KUKA KRL program: EPS_2_25862_MH4A_A_20251016034300.src

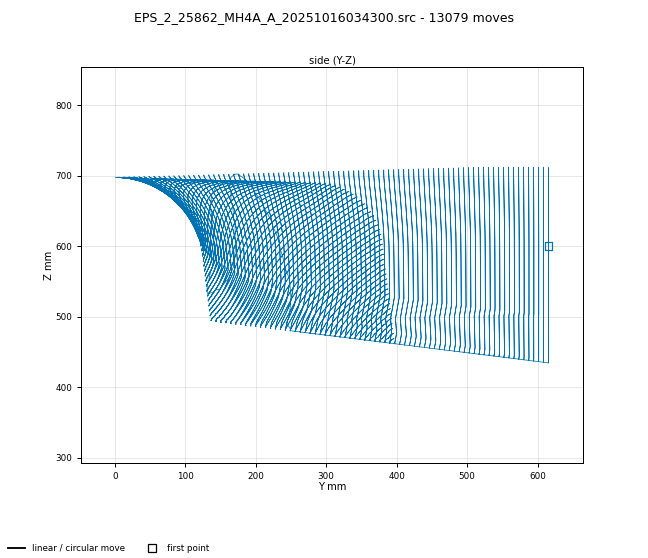
[picture p0: tool path of EPS_2_25862_MH4A_A_20251016034300.src, 13079 of 13081 moves have a stored position in this frame; points joined in program order, loops and branches not executed]
&ACCESS RVP
&REL 4
&COMMENT QRS 19112012
&PARAM EDITMASK = *
DEF PART()
EXT BAS (BAS_COMMAND :IN,REAL :IN )
INT I
BAS (#INITMOV,0 )

;KUKA QRS Post kuka4.cps  Date:22-06-2017 !

File_ID=2890

QRS_PRE_INIT()

;Init var - Until changes are made in qrs_pre_init
Outlet_Square_prg=0
Inlet_1_Square_prg=0
Inlet_2_Square_prg=0
Inlet_3_Square_prg=0
Inlet_4_Square_prg=0
Inlet_5_Square_prg=0

Outlet_1={X 0.000, Y 524.580, Z 611.500, B 0.000, E1 0.000 }
Inlet_1={X 0.000, Y 545.480, Z 586.500, B 0.000, E1 180.000 }
Outlet_1_type=201
Inlet_1_type=0
;QRS#1=Sidecore dimensions
;QRS#2=200-8" PVC SDR 35
;QRS#3=DeadEnd 201
;QRS#4=
;QRS#5=
;QRS#6=
;QRS#7=
;QRS#8=
;QRS#9=12-08 PSX
;QRS#10=

;QRS#11=
;QRS#12=
;QRS#13=
;QRS#14=
;QRS#15=
;QRS#16=1220x127x991 3,25'
;QRS#17=EPS Height
;QRS#18=712
;QRS#19=*
;QRS#20= UPDATED VERSION 22-06-2017
;QRS#21=*
Outlet_Square=0100
Inlet_1_Square=00
Inlet_2_Square=0
Inlet_3_Square=0
Inlet_4_Square=0
Inlet_5_Square=0
Mill_Square=1
Outlet_Square_Prg=204
Inlet_1_Square_prg=0

QRS_INIT()

$ADVANCE=5

; T1
PTP {E1 173.645,E2 173.645}
PTP {X 0,Y 615.456,A -85,B 0,C 180,E1 173.645,E2 173.645,E3 0,E4 0,E5 0,E6 0}
QRS_SPEED_INIT()
LIN {X 0,Y 615.456,Z 600,A -85,B 0,C 180,E1 173.645,E2 173.645,E3 0,E4 0,E5 0,E6 0} C_VEL
LIN {X 0,Y 615.456,Z 444.377,A -85,B 0,C 180,E1 173.645,E2 173.645} C_VEL
LIN {X 0,Y 615.456,Z 436.199,A -85,B 0,C 180,E1 173.645,E2 173.645} C_VEL
LIN {X 0,Y 615.435,Z 434.199,A -85,B 0,C 180,E1 173.459,E2 173.459} C_VEL
LIN {X 0,Y 615.436,Z 434.199,A -85,B 0,C 180,E1 171.464,E2 171.464} C_VEL
LIN {X 0,Y 615.416,Z 434.199,A -85,B 0,C 180,E1 169.144,E2 169.144} C_VEL
LIN {X 0,Y 615.415,Z 434.199,A -85,B 0,C 180,E1 166.798,E2 166.798} C_VEL
LIN {X 0,Y 615.478,Z 434.199,A -85,B 0,C 180,E1 164.096,E2 164.096} C_VEL
LIN {X 0,Y 615.426,Z 434.199,A -85,B 0,C 180,E1 161.353,E2 161.353} C_VEL
LIN {X 0,Y 615.42,Z 434.199,A -85,B 0,C 180,E1 159.268,E2 159.268} C_VEL
LIN {X 0,Y 615.415,Z 434.199,A -85,B 0,C 180,E1 157.154,E2 157.154} C_VEL
LIN {X 0,Y 615.412,Z 434.199,A -85,B 0,C 180,E1 155.006,E2 155.006} C_VEL
LIN {X 0,Y 615.414,Z 434.199,A -85,B 0,C 180,E1 152.821,E2 152.821} C_VEL
LIN {X 0,Y 615.467,Z 434.198,A -85,B 0,C 180,E1 150.208,E2 150.208} C_VEL
LIN {X 0,Y 615.441,Z 434.2,A -85,B 0,C 180,E1 147.541,E2 147.541} C_VEL
LIN {X 0,Y 615.415,Z 434.199,A -85,B 0,C 180,E1 145.182,E2 145.182} C_VEL
LIN {X 0,Y 615.416,Z 434.199,A -85,B 0,C 180,E1 142.755,E2 142.755} C_VEL
LIN {X 0,Y 615.492,Z 434.2,A -85,B 0,C 180,E1 139.91,E2 139.91} C_VEL
LIN {X 0,Y 615.452,Z 434.2,A -85,B 0,C 180,E1 137.646,E2 137.646} C_VEL
LIN {X 0,Y 615.411,Z 434.199,A -85,B 0,C 180,E1 135.075,E2 135.075} C_VEL
LIN {X 0,Y 615.411,Z 434.199,A -85,B 0,C 180,E1 133.042,E2 133.042} C_VEL
LIN {X 0,Y 615.423,Z 434.199,A -85,B 0,C 180,E1 130.611,E2 130.611} C_VEL
LIN {X 0,Y 615.472,Z 434.205,A -85,B 0,C 180,E1 128.013,E2 128.013} C_VEL
LIN {X 0,Y 615.447,Z 434.2,A -85,B 0,C 180,E1 125.618,E2 125.618} C_VEL
LIN {X 0,Y 615.416,Z 434.2,A -85,B 0,C 180,E1 123.24,E2 123.24} C_VEL
LIN {X 0,Y 615.41,Z 434.199,A -85,B 0,C 180,E1 120.924,E2 120.924} C_VEL
LIN {X 0,Y 615.437,Z 434.199,A -85,B 0,C 180,E1 118.445,E2 118.445} C_VEL
LIN {X 0,Y 615.439,Z 434.2,A -85,B 0,C 180,E1 115.563,E2 115.563} C_VEL
LIN {X 0,Y 615.439,Z 434.2,A -85,B 0,C 180,E1 113.558,E2 113.558} C_VEL
LIN {X 0,Y 615.427,Z 434.2,A -85,B 0,C 180,E1 111.434,E2 111.434} C_VEL
LIN {X 0,Y 615.42,Z 434.2,A -85,B 0,C 180,E1 109.34,E2 109.34} C_VEL
LIN {X 0,Y 615.416,Z 434.2,A -85,B 0,C 180,E1 107.272,E2 107.272} C_VEL
LIN {X 0,Y 615.413,Z 434.2,A -85,B 0,C 180,E1 105.228,E2 105.228} C_VEL
LIN {X 0,Y 615.411,Z 434.2,A -85,B 0,C 180,E1 103.203,E2 103.203} C_VEL
LIN {X 0,Y 615.409,Z 434.2,A -85,B 0,C 180,E1 100.859,E2 100.859} C_VEL
LIN {X 0,Y 615.428,Z 434.2,A -85,B 0,C 180,E1 98.537,E2 98.537} C_VEL
LIN {X 0,Y 615.481,Z 434.201,A -85,B 0,C 180,E1 95.899,E2 95.899} C_VEL
LIN {X 0,Y 615.414,Z 434.2,A -85,B 0,C 180,E1 93.273,E2 93.273} C_VEL
LIN {X 0,Y 615.416,Z 434.2,A -85,B 0,C 180,E1 91.309,E2 91.309} C_VEL
LIN {X 0,Y 615.418,Z 434.2,A -85,B 0,C 180,E1 89.346,E2 89.346} C_VEL
LIN {X 0,Y 615.421,Z 434.2,A -85,B 0,C 180,E1 87.382,E2 87.382} C_VEL
LIN {X 0,Y 615.424,Z 434.2,A -85,B 0,C 180,E1 85.415,E2 85.415} C_VEL
LIN {X 0,Y 615.425,Z 434.2,A -85,B 0,C 180,E1 83.443,E2 83.443} C_VEL
LIN {X 0,Y 615.428,Z 434.2,A -85,B 0,C 180,E1 81.463,E2 81.463} C_VEL
LIN {X 0,Y 615.409,Z 434.2,A -85,B 0,C 180,E1 79.141,E2 79.141} C_VEL
LIN {X 0,Y 615.411,Z 434.2,A -85,B 0,C 180,E1 76.797,E2 76.797} C_VEL
LIN {X 0,Y 615.478,Z 434.202,A -85,B 0,C 180,E1 74.095,E2 74.095} C_VEL
LIN {X 0,Y 615.42,Z 434.2,A -85,B 0,C 180,E1 71.352,E2 71.352} C_VEL
LIN {X 0,Y 615.415,Z 434.2,A -85,B 0,C 180,E1 69.267,E2 69.267} C_VEL
LIN {X 0,Y 615.411,Z 434.2,A -85,B 0,C 180,E1 67.153,E2 67.153} C_VEL
LIN {X 0,Y 615.409,Z 434.2,A -85,B 0,C 180,E1 65.005,E2 65.005} C_VEL
LIN {X 0,Y 615.471,Z 434.204,A -85,B 0,C 180,E1 62.084,E2 62.084} C_VEL
LIN {X 0,Y 615.474,Z 434.199,A -85,B 0,C 180,E1 59.84,E2 59.84} C_VEL
LIN {X 0,Y 615.436,Z 434.199,A -85,B 0,C 180,E1 57.54,E2 57.54} C_VEL
LIN {X 0,Y 615.412,Z 434.199,A -85,B 0,C 180,E1 55.181,E2 55.181} C_VEL
LIN {X 0,Y 615.416,Z 434.2,A -85,B 0,C 180,E1 52.753,E2 52.753} C_VEL
LIN {X 0,Y 615.485,Z 434.199,A -85,B 0,C 180,E1 49.909,E2 49.909} C_VEL
LIN {X 0,Y 615.447,Z 434.199,A -85,B 0,C 180,E1 47.644,E2 47.644} C_VEL
LIN {X 0,Y 615.411,Z 434.199,A -85,B 0,C 180,E1 45.074,E2 45.074} C_VEL
LIN {X 0,Y 615.411,Z 434.199,A -85,B 0,C 180,E1 43.04,E2 43.04} C_VEL
LIN {X 0,Y 615.411,Z 434.199,A -85,B 0,C 180,E1 41.087,E2 41.087} C_VEL
LIN {X 0,Y 615.412,Z 434.199,A -85,B 0,C 180,E1 38.908,E2 38.908} C_VEL
LIN {X 0,Y 615.444,Z 434.2,A -85,B 0,C 180,E1 36.426,E2 36.426} C_VEL
LIN {X 0,Y 615.435,Z 434.199,A -85,B 0,C 180,E1 33.528,E2 33.528} C_VEL
LIN {X 0,Y 615.412,Z 434.199,A -85,B 0,C 180,E1 30.922,E2 30.922} C_VEL
LIN {X 0,Y 615.443,Z 434.2,A -85,B 0,C 180,E1 28.444,E2 28.444} C_VEL
LIN {X 0,Y 615.439,Z 434.198,A -85,B 0,C 180,E1 25.561,E2 25.561} C_VEL
LIN {X 0,Y 615.438,Z 434.198,A -85,B 0,C 180,E1 23.557,E2 23.557} C_VEL
LIN {X 0,Y 615.428,Z 434.198,A -85,B 0,C 180,E1 21.433,E2 21.433} C_VEL
LIN {X 0,Y 615.421,Z 434.199,A -85,B 0,C 180,E1 19.339,E2 19.339} C_VEL
LIN {X 0,Y 615.417,Z 434.199,A -85,B 0,C 180,E1 17.271,E2 17.271} C_VEL
LIN {X 0,Y 615.416,Z 434.199,A -85,B 0,C 180,E1 15.227,E2 15.227} C_VEL
LIN {X 0,Y 615.415,Z 434.199,A -85,B 0,C 180,E1 13.202,E2 13.202} C_VEL
LIN {X 0,Y 615.416,Z 434.199,A -85,B 0,C 180,E1 10.856,E2 10.856} C_VEL
LIN {X 0,Y 615.436,Z 434.199,A -85,B 0,C 180,E1 8.536,E2 8.536} C_VEL
LIN {X 0,Y 615.481,Z 434.198,A -85,B 0,C 180,E1 5.898,E2 5.898} C_VEL
LIN {X 0,Y 615.419,Z 434.198,A -85,B 0,C 180,E1 3.272,E2 3.272} C_VEL
LIN {X 0,Y 615.42,Z 434.198,A -85,B 0,C 180,E1 1.308,E2 1.308} C_VEL
LIN {X 0,Y 615.423,Z 434.198,A -85,B 0,C 180,E1 -0.655,E2 -0.655} C_VEL
LIN {X 0,Y 615.425,Z 434.198,A -85,B 0,C 180,E1 -2.619,E2 -2.619} C_VEL
LIN {X 0,Y 615.427,Z 434.198,A -85,B 0,C 180,E1 -4.586,E2 -4.586} C_VEL
LIN {X 0,Y 615.429,Z 434.198,A -85,B 0,C 180,E1 -6.558,E2 -6.558} C_VEL
LIN {X 0,Y 615.431,Z 434.198,A -85,B 0,C 180,E1 -8.538,E2 -8.538} C_VEL
LIN {X 0,Y 615.415,Z 434.198,A -85,B 0,C 180,E1 -10.856,E2 -10.856} C_VEL
LIN {X 0,Y 615.42,Z 434.199,A -85,B 0,C 180,E1 -13.204,E2 -13.204} C_VEL
LIN {X 0,Y 615.482,Z 434.204,A -85,B 0,C 180,E1 -15.906,E2 -15.906} C_VEL
LIN {X 0,Y 615.424,Z 434.198,A -85,B 0,C 180,E1 -18.649,E2 -18.649} C_VEL
LIN {X 0,Y 615.42,Z 434.198,A -85,B 0,C 180,E1 -20.734,E2 -20.734} C_VEL
LIN {X 0,Y 615.416,Z 434.198,A -85,B 0,C 180,E1 -22.848,E2 -22.848} C_VEL
LIN {X 0,Y 615.416,Z 434.198,A -85,B 0,C 180,E1 -24.996,E2 -24.996} C_VEL
LIN {X 0,Y 615.477,Z 434.205,A -85,B 0,C 180,E1 -27.916,E2 -27.916} C_VEL
LIN {X 0,Y 615.474,Z 434.197,A -85,B 0,C 180,E1 -30.162,E2 -30.162} C_VEL
LIN {X 0,Y 615.438,Z 434.197,A -85,B 0,C 180,E1 -32.461,E2 -32.461} C_VEL
LIN {X 0,Y 615.417,Z 434.198,A -85,B 0,C 180,E1 -34.82,E2 -34.82} C_VEL
LIN {X 0,Y 615.416,Z 434.198,A -85,B 0,C 180,E1 -36.929,E2 -36.929} C_VEL
LIN {X 0,Y 615.417,Z 434.198,A -85,B 0,C 180,E1 -39.055,E2 -39.055} C_VEL
LIN {X 0,Y 615.442,Z 434.199,A -85,B 0,C 180,E1 -41.478,E2 -41.478} C_VEL
LIN {X 0,Y 615.476,Z 434.196,A -85,B 0,C 180,E1 -44.151,E2 -44.151} C_VEL
LIN {X 0,Y 615.42,Z 434.197,A -85,B 0,C 180,E1 -46.75,E2 -46.75} C_VEL
LIN {X 0,Y 615.417,Z 434.198,A -85,B 0,C 180,E1 -48.914,E2 -48.914} C_VEL
LIN {X 0,Y 615.419,Z 434.198,A -85,B 0,C 180,E1 -51.091,E2 -51.091} C_VEL
LIN {X 0,Y 615.455,Z 434.199,A -85,B 0,C 180,E1 -53.573,E2 -53.573} C_VEL
LIN {X 0,Y 615.438,Z 434.197,A -85,B 0,C 180,E1 -56.473,E2 -56.473} C_VEL
LIN {X 0,Y 615.419,Z 434.198,A -85,B 0,C 180,E1 -59.077,E2 -59.077} C_VEL
LIN {X 0,Y 615.453,Z 434.199,A -85,B 0,C 180,E1 -61.556,E2 -61.556} C_VEL
LIN {X 0,Y 615.441,Z 434.196,A -85,B 0,C 180,E1 -64.441,E2 -64.441} C_VEL
LIN {X 0,Y 615.497,Z 434.361,A -85,B 0,C 180,E1 -65.958,E2 -65.958} C_VEL
LIN {X 0,Y 615.49,Z 449.44,A -85,B 0,C 180,E1 -68.568,E2 -68.568} C_VEL
LIN {X 0,Y 615.488,Z 466.211,A -85,B 0,C 180,E1 -71.396,E2 -71.396} C_VEL
LIN {X 0,Y 615.484,Z 482.466,A -85,B 0,C 180,E1 -74.095,E2 -74.095} C_VEL
LIN {X 0,Y 615.496,Z 498.953,A -85,B 0,C 180,E1 -76.799,E2 -76.799} C_VEL
LIN {X 0,Y 615.471,Z 501.196,A -85,B 0,C 180,E1 -77.113,E2 -77.113} C_VEL
LIN {X 0,Y 615.468,Z 503.698,A -85,B 0,C 180,E1 -77.176,E2 -77.176} C_VEL
LIN {X 0,Y 615.497,Z 607.835,A -85,B 0,C 180,E1 -78.411,E2 -78.411} C_VEL
LIN {X 0,Y 615.499,Z 620.346,A -85,B 0,C 180,E1 -78.682,E2 -78.682} C_VEL
LIN {X 0,Y 615.496,Z 633.505,A -85,B 0,C 180,E1 -79.109,E2 -79.109} C_VEL
LIN {X 0,Y 615.493,Z 645.478,A -85,B 0,C 180,E1 -79.64,E2 -79.64} C_VEL
LIN {X 0,Y 615.492,Z 656.996,A -85,B 0,C 180,E1 -80.304,E2 -80.304} C_VEL
LIN {X 0,Y 615.499,Z 667.342,A -85,B 0,C 180,E1 -81.05,E2 -81.05} C_VEL
LIN {X 0,Y 615.497,Z 675.813,A -85,B 0,C 180,E1 -81.794,E2 -81.794} C_VEL
LIN {X 0,Y 615.498,Z 683.607,A -85,B 0,C 180,E1 -82.62,E2 -82.62} C_VEL
LIN {X 0,Y 615.496,Z 691.203,A -85,B 0,C 180,E1 -83.608,E2 -83.608} C_VEL
LIN {X 0,Y 615.498,Z 698.205,A -85,B 0,C 180,E1 -84.759,E2 -84.759} C_VEL
LIN {X 0,Y 615.494,Z 702.851,A -85,B 0,C 180,E1 -85.744,E2 -85.744} C_VEL
LIN {X 0,Y 615.494,Z 706.399,A -85,B 0,C 180,E1 -86.727,E2 -86.727} C_VEL
LIN {X 0,Y 615.497,Z 708.233,A -85,B 0,C 180,E1 -87.382,E2 -87.382} C_VEL
LIN {X 0,Y 615.499,Z 709.608,A -85,B 0,C 180,E1 -88.037,E2 -88.037} C_VEL
LIN {X 0,Y 615.496,Z 711.174,A -85,B 0,C 180,E1 -89.346,E2 -89.346} C_VEL
LIN {X 0,Y 615.494,Z 711.389,A -85,B 0,C 180,E1 -90,E2 -90} C_VEL
LIN {X 0,Y 615.495,Z 710.58,A -85,B 0,C 180,E1 -91.309,E2 -91.309} C_VEL
LIN {X 0,Y 615.499,Z 709.608,A -85,B 0,C 180,E1 -91.963,E2 -91.963} C_VEL
LIN {X 0,Y 615.497,Z 708.233,A -85,B 0,C 180,E1 -92.618,E2 -92.618} C_VEL
LIN {X 0,Y 615.496,Z 705.35,A -85,B 0,C 180,E1 -93.601,E2 -93.601} C_VEL
LIN {X 0,Y 615.498,Z 701.442,A -85,B 0,C 180,E1 -94.584,E2 -94.584} C_VEL
LIN {X 0,Y 615.499,Z 696.405,A -85,B 0,C 180,E1 -95.57,E2 -95.57} C_VEL
LIN {X 0,Y 615.497,Z 689.871,A -85,B 0,C 180,E1 -96.583,E2 -96.583} C_VEL
LIN {X 0,Y 615.497,Z 682.134,A -85,B 0,C 180,E1 -97.545,E2 -97.545} C_VEL
LIN {X 0,Y 615.498,Z 674.046,A -85,B 0,C 180,E1 -98.371,E2 -98.371} C_VEL
LIN {X 0,Y 615.499,Z 664.169,A -85,B 0,C 180,E1 -99.199,E2 -99.199} C_VEL
LIN {X 0,Y 615.492,Z 652.982,A -85,B 0,C 180,E1 -99.945,E2 -99.945} C_VEL
LIN {X 0,Y 615.494,Z 642.024,A -85,B 0,C 180,E1 -100.527,E2 -100.527} C_VEL
LIN {X 0,Y 615.499,Z 629.422,A -85,B 0,C 180,E1 -101.042,E2 -101.042} C_VEL
LIN {X 0,Y 615.499,Z 617.068,A -85,B 0,C 180,E1 -101.401,E2 -101.401} C_VEL
LIN {X 0,Y 615.498,Z 603.472,A -85,B 0,C 180,E1 -101.652,E2 -101.652} C_VEL
LIN {X 0,Y 615.47,Z 501.548,A -85,B 0,C 180,E1 -102.866,E2 -102.866} C_VEL
LIN {X 0,Y 615.48,Z 499.988,A -85,B 0,C 180,E1 -103.033,E2 -103.033} C_VEL
LIN {X 0,Y 615.473,Z 483.5,A -85,B 0,C 180,E1 -105.735,E2 -105.735} C_VEL
LIN {X 0,Y 615.488,Z 468.149,A -85,B 0,C 180,E1 -108.28,E2 -108.28} C_VEL
LIN {X 0,Y 615.461,Z 451.507,A -85,B 0,C 180,E1 -111.082,E2 -111.082} C_VEL
LIN {X 0,Y 615.497,Z 435.726,A -85,B 0,C 180,E1 -113.782,E2 -113.782} C_VEL
LIN {X 0,Y 615.498,Z 434.288,A -85,B 0,C 180,E1 -114.075,E2 -114.075} C_VEL
LIN {X 0,Y 615.453,Z 434.199,A -85,B 0,C 180,E1 -116.445,E2 -116.445} C_VEL
LIN {X 0,Y 615.433,Z 434.199,A -85,B 0,C 180,E1 -118.66,E2 -118.66} C_VEL
LIN {X 0,Y 615.418,Z 434.198,A -85,B 0,C 180,E1 -121.074,E2 -121.074} C_VEL
LIN {X 0,Y 615.438,Z 434.197,A -85,B 0,C 180,E1 -123.526,E2 -123.526} C_VEL
LIN {X 0,Y 615.455,Z 434.199,A -85,B 0,C 180,E1 -126.427,E2 -126.427} C_VEL
LIN {X 0,Y 615.419,Z 434.198,A -85,B 0,C 180,E1 -128.909,E2 -128.909} C_VEL
LIN {X 0,Y 615.417,Z 434.198,A -85,B 0,C 180,E1 -131.086,E2 -131.086} C_VEL
LIN {X 0,Y 615.42,Z 434.197,A -85,B 0,C 180,E1 -133.25,E2 -133.25} C_VEL
LIN {X 0,Y 615.476,Z 434.196,A -85,B 0,C 180,E1 -135.849,E2 -135.849} C_VEL
LIN {X 0,Y 615.442,Z 434.199,A -85,B 0,C 180,E1 -138.522,E2 -138.522} C_VEL
LIN {X 0,Y 615.417,Z 434.198,A -85,B 0,C 180,E1 -140.945,E2 -140.945} C_VEL
LIN {X 0,Y 615.416,Z 434.198,A -85,B 0,C 180,E1 -143.071,E2 -143.071} C_VEL
LIN {X 0,Y 615.421,Z 434.198,A -85,B 0,C 180,E1 -145.307,E2 -145.307} C_VEL
LIN {X 0,Y 615.45,Z 434.197,A -85,B 0,C 180,E1 -147.674,E2 -147.674} C_VEL
LIN {X 0,Y 615.435,Z 434.199,A -85,B 0,C 180,E1 -150.59,E2 -150.59} C_VEL
LIN {X 0,Y 615.416,Z 434.198,A -85,B 0,C 180,E1 -152.967,E2 -152.967} C_VEL
LIN {X 0,Y 615.416,Z 434.198,A -85,B 0,C 180,E1 -155.004,E2 -155.004} C_VEL
LIN {X 0,Y 615.416,Z 434.198,A -85,B 0,C 180,E1 -157.152,E2 -157.152} C_VEL
LIN {X 0,Y 615.481,Z 434.2,A -85,B 0,C 180,E1 -159.966,E2 -159.966} C_VEL
LIN {X 0,Y 615.423,Z 434.199,A -85,B 0,C 180,E1 -162.727,E2 -162.727} C_VEL
LIN {X 0,Y 615.422,Z 434.199,A -85,B 0,C 180,E1 -164.771,E2 -164.771} C_VEL
LIN {X 0,Y 615.419,Z 434.199,A -85,B 0,C 180,E1 -166.796,E2 -166.796} C_VEL
LIN {X 0,Y 615.415,Z 434.198,A -85,B 0,C 180,E1 -169.144,E2 -169.144} C_VEL
LIN {X 0,Y 615.431,Z 434.198,A -85,B 0,C 180,E1 -171.462,E2 -171.462} C_VEL
LIN {X 0,Y 615.493,Z 434.201,A -85,B 0,C 180,E1 -174.101,E2 -174.101} C_VEL
LIN {X 0,Y 615.423,Z 434.199,A -85,B 0,C 180,E1 -176.726,E2 -176.726} C_VEL
LIN {X 0,Y 615.425,Z 434.199,A -85,B 0,C 180,E1 -178.69,E2 -178.69} C_VEL
LIN {X 0,Y 615.427,Z 434.199,A -85,B 0,C 180,E1 -180.653,E2 -180.653} C_VEL
LIN {X 0,Y 615.43,Z 434.199,A -85,B 0,C 180,E1 -182.617,E2 -182.617} C_VEL
LIN {X 0,Y 615.432,Z 434.199,A -85,B 0,C 180,E1 -184.584,E2 -184.584} C_VEL
LIN {X 0,Y 615.435,Z 434.199,A -85,B 0,C 180,E1 -186.541,E2 -186.541} C_VEL
LIN {X 0,Y 614.743,Z 434.344,A -85,B 0,C 180,E1 -187.087,E2 -187.087} C_VEL
LIN {X 0,Y 611.895,Z 434.768,A -85,B 0,C 180,E1 -187.973,E2 -187.973} C_VEL
LIN {X 0,Y 609.51,Z 435.07,A -85,B 0,C 180,E1 -188.686,E2 -188.686} C_VEL
LIN {X 0,Y 608.493,Z 435.184,A -85,B 0,C 180,E1 -189.236,E2 -189.236} C_VEL
LIN {X 0,Y 608.412,Z 435.193,A -85,B 0,C 180,E1 -189.422,E2 -189.422} C_VEL
LIN {X 0,Y 608.445,Z 435.198,A -85,B 0,C 180,E1 -191.999,E2 -191.999} C_VEL
LIN {X 0,Y 608.392,Z 435.196,A -85,B 0,C 180,E1 -194.721,E2 -194.721} C_VEL
LIN {X 0,Y 608.4,Z 435.194,A -85,B 0,C 180,E1 -196.784,E2 -196.784} C_VEL
LIN {X 0,Y 608.39,Z 435.195,A -85,B 0,C 180,E1 -198.87,E2 -198.87} C_VEL
LIN {X 0,Y 608.405,Z 435.193,A -85,B 0,C 180,E1 -200.982,E2 -200.982} C_VEL
LIN {X 0,Y 608.454,Z 435.194,A -85,B 0,C 180,E1 -203.844,E2 -203.844} C_VEL
LIN {X 0,Y 608.41,Z 435.203,A -85,B 0,C 180,E1 -206.036,E2 -206.036} C_VEL
LIN {X 0,Y 608.399,Z 435.196,A -85,B 0,C 180,E1 -208.608,E2 -208.608} C_VEL
LIN {X 0,Y 608.414,Z 435.195,A -85,B 0,C 180,E1 -210.546,E2 -210.546} C_VEL
LIN {X 0,Y 608.406,Z 435.193,A -85,B 0,C 180,E1 -212.881,E2 -212.881} C_VEL
LIN {X 0,Y 608.395,Z 435.195,A -85,B 0,C 180,E1 -215.279,E2 -215.279} C_VEL
LIN {X 0,Y 608.449,Z 435.195,A -85,B 0,C 180,E1 -218.239,E2 -218.239} C_VEL
LIN {X 0,Y 608.426,Z 435.196,A -85,B 0,C 180,E1 -220.327,E2 -220.327} C_VEL
LIN {X 0,Y 608.425,Z 435.196,A -85,B 0,C 180,E1 -222.331,E2 -222.331} C_VEL
LIN {X 0,Y 608.394,Z 435.195,A -85,B 0,C 180,E1 -224.799,E2 -224.799} C_VEL
LIN {X 0,Y 608.381,Z 435.195,A -85,B 0,C 180,E1 -227.034,E2 -227.034} C_VEL
LIN {X 0,Y 608.385,Z 435.196,A -85,B 0,C 180,E1 -228.818,E2 -228.818} C_VEL
LIN {X 0,Y 608.39,Z 435.196,A -85,B 0,C 180,E1 -231.407,E2 -231.407} C_VEL
LIN {X 0,Y 608.43,Z 435.2,A -85,B 0,C 180,E1 -233.954,E2 -233.954} C_VEL
LIN {X 0,Y 608.426,Z 435.196,A -85,B 0,C 180,E1 -236.327,E2 -236.327} C_VEL
LIN {X 0,Y 608.41,Z 435.193,A -85,B 0,C 180,E1 -238.735,E2 -238.735} C_VEL
LIN {X 0,Y 608.381,Z 435.196,A -85,B 0,C 180,E1 -240.976,E2 -240.976} C_VEL
LIN {X 0,Y 608.384,Z 435.196,A -85,B 0,C 180,E1 -243.223,E2 -243.223} C_VEL
LIN {X 0,Y 608.443,Z 435.196,A -85,B 0,C 180,E1 -245.851,E2 -245.851} C_VEL
LIN {X 0,Y 608.431,Z 435.196,A -85,B 0,C 180,E1 -248.307,E2 -248.307} C_VEL
LIN {X 0,Y 608.408,Z 435.193,A -85,B 0,C 180,E1 -251.129,E2 -251.129} C_VEL
LIN {X 0,Y 608.438,Z 435.198,A -85,B 0,C 180,E1 -253.906,E2 -253.906} C_VEL
LIN {X 0,Y 608.408,Z 435.194,A -85,B 0,C 180,E1 -256.642,E2 -256.642} C_VEL
LIN {X 0,Y 608.379,Z 435.196,A -85,B 0,C 180,E1 -259.079,E2 -259.079} C_VEL
LIN {X 0,Y 608.4,Z 435.195,A -85,B 0,C 180,E1 -261.363,E2 -261.363} C_VEL
LIN {X 0,Y 608.448,Z 435.199,A -85,B 0,C 180,E1 -264.033,E2 -264.033} C_VEL
LIN {X 0,Y 608.387,Z 435.196,A -85,B 0,C 180,E1 -266.689,E2 -266.689} C_VEL
LIN {X 0,Y 608.407,Z 435.194,A -85,B 0,C 180,E1 -268.676,E2 -268.676} C_VEL
LIN {X 0,Y 608.396,Z 435.195,A -85,B 0,C 180,E1 -270.662,E2 -270.662} C_VEL
LIN {X 0,Y 608.416,Z 435.193,A -85,B 0,C 180,E1 -272.648,E2 -272.648} C_VEL
LIN {X 0,Y 608.402,Z 435.195,A -85,B 0,C 180,E1 -275.302,E2 -275.302} C_VEL
LIN {X 0,Y 608.459,Z 435.197,A -85,B 0,C 180,E1 -277.967,E2 -277.967} C_VEL
LIN {X 0,Y 608.402,Z 435.195,A -85,B 0,C 180,E1 -280.651,E2 -280.651} C_VEL
LIN {X 0,Y 608.391,Z 435.196,A -85,B 0,C 180,E1 -282.679,E2 -282.679} C_VEL
LIN {X 0,Y 608.386,Z 435.196,A -85,B 0,C 180,E1 -284.723,E2 -284.723} C_VEL
LIN {X 0,Y 608.394,Z 435.195,A -85,B 0,C 180,E1 -286.786,E2 -286.786} C_VEL
LIN {X 0,Y 608.408,Z 435.193,A -85,B 0,C 180,E1 -288.871,E2 -288.871} C_VEL
LIN {X 0,Y 608.431,Z 435.196,A -85,B 0,C 180,E1 -291.693,E2 -291.693} C_VEL
LIN {X 0,Y 608.408,Z 435.194,A -85,B 0,C 180,E1 -294.573,E2 -294.573} C_VEL
LIN {X 0,Y 608.395,Z 435.195,A -85,B 0,C 180,E1 -297.196,E2 -297.196} C_VEL
LIN {X 0,Y 608.452,Z 435.198,A -85,B 0,C 180,E1 -299.972,E2 -299.972} C_VEL
LIN {X 0,Y 608.403,Z 435.193,A -85,B 0,C 180,E1 -302.882,E2 -302.882} C_VEL
LIN {X 0,Y 608.395,Z 435.195,A -85,B 0,C 180,E1 -305.28,E2 -305.28} C_VEL
LIN {X 0,Y 608.445,Z 435.194,A -85,B 0,C 180,E1 -308.24,E2 -308.24} C_VEL
LIN {X 0,Y 608.421,Z 435.195,A -85,B 0,C 180,E1 -310.328,E2 -310.328} C_VEL
LIN {X 0,Y 608.42,Z 435.195,A -85,B 0,C 180,E1 -312.332,E2 -312.332} C_VEL
LIN {X 0,Y 608.393,Z 435.195,A -85,B 0,C 180,E1 -314.801,E2 -314.801} C_VEL
LIN {X 0,Y 608.382,Z 435.196,A -85,B 0,C 180,E1 -317.036,E2 -317.036} C_VEL
LIN {X 0,Y 608.384,Z 435.196,A -85,B 0,C 180,E1 -318.82,E2 -318.82} C_VEL
LIN {X 0,Y 608.392,Z 435.197,A -85,B 0,C 180,E1 -321.408,E2 -321.408} C_VEL
LIN {X 0,Y 608.431,Z 435.201,A -85,B 0,C 180,E1 -323.956,E2 -323.956} C_VEL
LIN {X 0,Y 608.43,Z 435.194,A -85,B 0,C 180,E1 -326.329,E2 -326.329} C_VEL
LIN {X 0,Y 608.413,Z 435.193,A -85,B 0,C 180,E1 -328.737,E2 -328.737} C_VEL
LIN {X 0,Y 608.384,Z 435.195,A -85,B 0,C 180,E1 -330.977,E2 -330.977} C_VEL
LIN {X 0,Y 608.388,Z 435.195,A -85,B 0,C 180,E1 -333.224,E2 -333.224} C_VEL
LIN {X 0,Y 608.451,Z 435.197,A -85,B 0,C 180,E1 -335.852,E2 -335.852} C_VEL
LIN {X 0,Y 608.435,Z 435.194,A -85,B 0,C 180,E1 -338.309,E2 -338.309} C_VEL
LIN {X 0,Y 608.412,Z 435.195,A -85,B 0,C 180,E1 -340.429,E2 -340.429} C_VEL
LIN {X 0,Y 608.408,Z 435.194,A -85,B 0,C 180,E1 -342.523,E2 -342.523} C_VEL
LIN {X 0,Y 608.422,Z 435.192,A -85,B 0,C 180,E1 -344.594,E2 -344.594} C_VEL
LIN {X 0,Y 608.411,Z 435.193,A -85,B 0,C 180,E1 -346.644,E2 -346.644} C_VEL
LIN {X 0,Y 608.385,Z 435.195,A -85,B 0,C 180,E1 -349.082,E2 -349.082} C_VEL
LIN {X 0,Y 608.408,Z 435.194,A -85,B 0,C 180,E1 -351.364,E2 -351.364} C_VEL
LIN {X 0,Y 608.45,Z 435.197,A -85,B 0,C 180,E1 -354.034,E2 -354.034} C_VEL
LIN {X 0,Y 608.391,Z 435.195,A -85,B 0,C 180,E1 -356.69,E2 -356.69} C_VEL
LIN {X 0,Y 608.411,Z 435.192,A -85,B 0,C 180,E1 -358.677,E2 -358.677} C_VEL
LIN {X 0,Y 608.401,Z 435.194,A -85,B 0,C 180,E1 -360.663,E2 -360.663} C_VEL
LIN {X 0,Y 608.421,Z 435.192,A -85,B 0,C 180,E1 -362.649,E2 -362.649} C_VEL
LIN {X 0,Y 608.411,Z 435.194,A -85,B 0,C 180,E1 -365.303,E2 -365.303} C_VEL
LIN {X 0,Y 608.467,Z 435.195,A -85,B 0,C 180,E1 -367.968,E2 -367.968} C_VEL
LIN {X 0,Y 608.407,Z 435.193,A -85,B 0,C 180,E1 -370.652,E2 -370.652} C_VEL
LIN {X 0,Y 608.396,Z 435.195,A -85,B 0,C 180,E1 -372.679,E2 -372.679} C_VEL
LIN {X 0,Y 608.392,Z 435.195,A -85,B 0,C 180,E1 -374.723,E2 -374.723} C_VEL
LIN {X 0,Y 608.401,Z 435.193,A -85,B 0,C 180,E1 -376.786,E2 -376.786} C_VEL
LIN {X 0,Y 608.393,Z 435.194,A -85,B 0,C 180,E1 -378.872,E2 -378.872} C_VEL
LIN {X 0,Y 608.409,Z 435.192,A -85,B 0,C 180,E1 -380.984,E2 -380.984} C_VEL
LIN {X 0,Y 608.455,Z 435.197,A -85,B 0,C 180,E1 -383.846,E2 -383.846} C_VEL
LIN {X 0,Y 608.418,Z 435.2,A -85,B 0,C 180,E1 -386.038,E2 -386.038} C_VEL
LIN {X 0,Y 608.398,Z 435.195,A -85,B 0,C 180,E1 -388.608,E2 -388.608} C_VEL
LIN {X 0,Y 608.413,Z 435.193,A -85,B 0,C 180,E1 -390.549,E2 -390.549} C_VEL
LIN {X 0,Y 608.41,Z 435.192,A -85,B 0,C 180,E1 -392.883,E2 -392.883} C_VEL
LIN {X 0,Y 608.403,Z 435.195,A -85,B 0,C 180,E1 -395.281,E2 -395.281} C_VEL
LIN {X 0,Y 608.424,Z 435.195,A -85,B 0,C 180,E1 -398.236,E2 -398.236} C_VEL
LIN {X 0,Y 608.432,Z 435.193,A -85,B 0,C 180,E1 -400.328,E2 -400.328} C_VEL
LIN {X 0,Y 608.423,Z 435.194,A -85,B 0,C 180,E1 -402.331,E2 -402.331} C_VEL
LIN {X 0,Y 608.399,Z 435.194,A -85,B 0,C 180,E1 -404.802,E2 -404.802} C_VEL
LIN {X 0,Y 608.389,Z 435.195,A -85,B 0,C 180,E1 -407.035,E2 -407.035} C_VEL
LIN {X 0,Y 608.39,Z 435.195,A -85,B 0,C 180,E1 -408.819,E2 -408.819} C_VEL
LIN {X 0,Y 608.4,Z 435.197,A -85,B 0,C 180,E1 -411.407,E2 -411.407} C_VEL
LIN {X 0,Y 608.441,Z 435.198,A -85,B 0,C 180,E1 -413.956,E2 -413.956} C_VEL
LIN {X 0,Y 608.444,Z 435.192,A -85,B 0,C 180,E1 -416.328,E2 -416.328} C_VEL
LIN {X 0,Y 608.405,Z 435.193,A -85,B 0,C 180,E1 -418.74,E2 -418.74} C_VEL
LIN {X 0,Y 608.391,Z 435.195,A -85,B 0,C 180,E1 -420.976,E2 -420.976} C_VEL
LIN {X 0,Y 608.397,Z 435.196,A -85,B 0,C 180,E1 -423.224,E2 -423.224} C_VEL
LIN {X 0,Y 608.491,Z 435.335,A -85,B 0,C 180,E1 -425.846,E2 -425.846} C_VEL
LIN {X 0,Y 608.544,Z 449.463,A -85,B 0,C 180,E1 -428.312,E2 -428.312} C_VEL
LIN {X 0,Y 608.515,Z 466.851,A -85,B 0,C 180,E1 -431.273,E2 -431.273} C_VEL
LIN {X 0,Y 608.49,Z 483.611,A -85,B 0,C 180,E1 -434.079,E2 -434.079} C_VEL
LIN {X 0,Y 608.469,Z 500.721,A -85,B 0,C 180,E1 -436.899,E2 -436.899} C_VEL
LIN {X 0,Y 608.484,Z 501.58,A -85,B 0,C 180,E1 -436.984,E2 -436.984} C_VEL
LIN {X 0,Y 608.56,Z 525.196,A -85,B 0,C 180,E1 -437.283,E2 -437.283} C_VEL
LIN {X 0,Y 608.549,Z 607.947,A -85,B 0,C 180,E1 -438.277,E2 -438.277} C_VEL
LIN {X 0,Y 608.548,Z 621.226,A -85,B 0,C 180,E1 -438.572,E2 -438.572} C_VEL
LIN {X 0,Y 608.54,Z 634.397,A -85,B 0,C 180,E1 -439.011,E2 -439.011} C_VEL
LIN {X 0,Y 608.512,Z 645.628,A -85,B 0,C 180,E1 -439.519,E2 -439.519} C_VEL
LIN {X 0,Y 608.483,Z 657.195,A -85,B 0,C 180,E1 -440.191,E2 -440.191} C_VEL
LIN {X 0,Y 608.485,Z 667.593,A -85,B 0,C 180,E1 -440.946,E2 -440.946} C_VEL
LIN {X 0,Y 608.475,Z 676.112,A -85,B 0,C 180,E1 -441.699,E2 -441.699} C_VEL
LIN {X 0,Y 608.471,Z 683.961,A -85,B 0,C 180,E1 -442.534,E2 -442.534} C_VEL
LIN {X 0,Y 608.461,Z 691.287,A -85,B 0,C 180,E1 -443.485,E2 -443.485} C_VEL
LIN {X 0,Y 608.45,Z 696.865,A -85,B 0,C 180,E1 -444.366,E2 -444.366} C_VEL
LIN {X 0,Y 608.432,Z 701.948,A -85,B 0,C 180,E1 -445.362,E2 -445.362} C_VEL
LIN {X 0,Y 608.449,Z 705.895,A -85,B 0,C 180,E1 -446.358,E2 -446.358} C_VEL
LIN {X 0,Y 608.425,Z 708.809,A -85,B 0,C 180,E1 -447.352,E2 -447.352} C_VEL
LIN {X 0,Y 608.444,Z 710.202,A -85,B 0,C 180,E1 -448.014,E2 -448.014} C_VEL
LIN {X 0,Y 608.438,Z 711.784,A -85,B 0,C 180,E1 -449.338,E2 -449.338} C_VEL
LIN {X 0,Y 608.434,Z 712,A -85,B 0,C 180,E1 -450,E2 -450} C_VEL
LIN {X 0,Y 608.448,Z 711.184,A -85,B 0,C 180,E1 -451.324,E2 -451.324} C_VEL
LIN {X 0,Y 608.444,Z 710.202,A -85,B 0,C 180,E1 -451.986,E2 -451.986} C_VEL
LIN {X 0,Y 608.425,Z 708.809,A -85,B 0,C 180,E1 -452.648,E2 -452.648} C_VEL
LIN {X 0,Y 608.449,Z 705.895,A -85,B 0,C 180,E1 -453.642,E2 -453.642} C_VEL
LIN {X 0,Y 608.432,Z 701.948,A -85,B 0,C 180,E1 -454.638,E2 -454.638} C_VEL
LIN {X 0,Y 608.437,Z 695.878,A -85,B 0,C 180,E1 -455.801,E2 -455.801} C_VEL
LIN {X 0,Y 608.462,Z 689.236,A -85,B 0,C 180,E1 -456.799,E2 -456.799} C_VEL
LIN {X 0,Y 608.456,Z 680.99,A -85,B 0,C 180,E1 -457.8,E2 -457.8} C_VEL
LIN {X 0,Y 608.472,Z 672.534,A -85,B 0,C 180,E1 -458.636,E2 -458.636} C_VEL
LIN {X 0,Y 608.478,Z 662.093,A -85,B 0,C 180,E1 -459.473,E2 -459.473} C_VEL
LIN {X 0,Y 608.503,Z 651.759,A -85,B 0,C 180,E1 -460.144,E2 -460.144} C_VEL
LIN {X 0,Y 608.523,Z 640.239,A -85,B 0,C 180,E1 -460.741,E2 -460.741} C_VEL
LIN {X 0,Y 608.533,Z 628.868,A -85,B 0,C 180,E1 -461.192,E2 -461.192} C_VEL
LIN {X 0,Y 608.551,Z 616.268,A -85,B 0,C 180,E1 -461.554,E2 -461.554} C_VEL
LIN {X 0,Y 608.548,Z 603.61,A -85,B 0,C 180,E1 -461.787,E2 -461.787} C_VEL
LIN {X 0,Y 608.547,Z 502.261,A -85,B 0,C 180,E1 -462.993,E2 -462.993} C_VEL
LIN {X 0,Y 608.459,Z 501.031,A -85,B 0,C 180,E1 -463.059,E2 -463.059} C_VEL
LIN {X 0,Y 608.442,Z 485.681,A -85,B 0,C 180,E1 -465.578,E2 -465.578} C_VEL
LIN {X 0,Y 608.488,Z 470.159,A -85,B 0,C 180,E1 -468.17,E2 -468.17} C_VEL
LIN {X 0,Y 608.478,Z 455.357,A -85,B 0,C 180,E1 -470.68,E2 -470.68} C_VEL
LIN {X 0,Y 608.551,Z 440.15,A -85,B 0,C 180,E1 -473.3,E2 -473.3} C_VEL
LIN {X 0,Y 608.473,Z 435.297,A -85,B 0,C 180,E1 -474.198,E2 -474.198} C_VEL
LIN {X 0,Y 608.397,Z 435.196,A -85,B 0,C 180,E1 -476.776,E2 -476.776} C_VEL
LIN {X 0,Y 608.391,Z 435.195,A -85,B 0,C 180,E1 -479.024,E2 -479.024} C_VEL
LIN {X 0,Y 608.407,Z 435.193,A -85,B 0,C 180,E1 -481.32,E2 -481.32} C_VEL
LIN {X 0,Y 608.447,Z 435.192,A -85,B 0,C 180,E1 -483.731,E2 -483.731} C_VEL
LIN {X 0,Y 608.439,Z 435.2,A -85,B 0,C 180,E1 -486.092,E2 -486.092} C_VEL
LIN {X 0,Y 608.4,Z 435.197,A -85,B 0,C 180,E1 -488.593,E2 -488.593} C_VEL
LIN {X 0,Y 608.39,Z 435.195,A -85,B 0,C 180,E1 -491.181,E2 -491.181} C_VEL
LIN {X 0,Y 608.417,Z 435.192,A -85,B 0,C 180,E1 -493.303,E2 -493.303} C_VEL
LIN {X 0,Y 608.458,Z 435.197,A -85,B 0,C 180,E1 -496.129,E2 -496.129} C_VEL
LIN {X 0,Y 608.392,Z 435.195,A -85,B 0,C 180,E1 -498.818,E2 -498.818} C_VEL
LIN {X 0,Y 608.395,Z 435.195,A -85,B 0,C 180,E1 -501.406,E2 -501.406} C_VEL
LIN {X 0,Y 608.442,Z 435.197,A -85,B 0,C 180,E1 -503.954,E2 -503.954} C_VEL
LIN {X 0,Y 608.441,Z 435.195,A -85,B 0,C 180,E1 -506.327,E2 -506.327} C_VEL
LIN {X 0,Y 608.421,Z 435.192,A -85,B 0,C 180,E1 -508.735,E2 -508.735} C_VEL
LIN {X 0,Y 608.389,Z 435.195,A -85,B 0,C 180,E1 -510.975,E2 -510.975} C_VEL
LIN {X 0,Y 608.39,Z 435.195,A -85,B 0,C 180,E1 -513.222,E2 -513.222} C_VEL
LIN {X 0,Y 608.447,Z 435.194,A -85,B 0,C 180,E1 -515.853,E2 -515.853} C_VEL
LIN {X 0,Y 608.438,Z 435.196,A -85,B 0,C 180,E1 -518.307,E2 -518.307} C_VEL
LIN {X 0,Y 608.417,Z 435.196,A -85,B 0,C 180,E1 -520.427,E2 -520.427} C_VEL
LIN {X 0,Y 608.416,Z 435.195,A -85,B 0,C 180,E1 -522.522,E2 -522.522} C_VEL
LIN {X 0,Y 608.427,Z 435.193,A -85,B 0,C 180,E1 -524.592,E2 -524.592} C_VEL
LIN {X 0,Y 608.417,Z 435.194,A -85,B 0,C 180,E1 -526.642,E2 -526.642} C_VEL
LIN {X 0,Y 608.386,Z 435.195,A -85,B 0,C 180,E1 -529.082,E2 -529.082} C_VEL
LIN {X 0,Y 608.405,Z 435.193,A -85,B 0,C 180,E1 -531.362,E2 -531.362} C_VEL
LIN {X 0,Y 608.459,Z 435.197,A -85,B 0,C 180,E1 -534.032,E2 -534.032} C_VEL
LIN {X 0,Y 608.395,Z 435.196,A -85,B 0,C 180,E1 -536.688,E2 -536.688} C_VEL
LIN {X 0,Y 608.415,Z 435.193,A -85,B 0,C 180,E1 -538.675,E2 -538.675} C_VEL
LIN {X 0,Y 608.405,Z 435.194,A -85,B 0,C 180,E1 -540.661,E2 -540.661} C_VEL
LIN {X 0,Y 608.424,Z 435.192,A -85,B 0,C 180,E1 -542.647,E2 -542.647} C_VEL
LIN {X 0,Y 608.406,Z 435.193,A -85,B 0,C 180,E1 -545.301,E2 -545.301} C_VEL
LIN {X 0,Y 608.463,Z 435.195,A -85,B 0,C 180,E1 -547.966,E2 -547.966} C_VEL
LIN {X 0,Y 608.412,Z 435.193,A -85,B 0,C 180,E1 -549.422,E2 -549.422} C_VEL
LIN {X 0,Y 607.758,Z 435.283,A -85,B 0,C 180,E1 -549.974,E2 -549.974} C_VEL
LIN {X 0,Y 604.928,Z 435.639,A -85,B 0,C 180,E1 -550.871,E2 -550.871} C_VEL
LIN {X 0,Y 602.519,Z 435.94,A -85,B 0,C 180,E1 -551.593,E2 -551.593} C_VEL
LIN {X 0,Y 601.466,Z 436.067,A -85,B 0,C 180,E1 -552.149,E2 -552.149} C_VEL
LIN {X 0,Y 601.37,Z 436.075,A -85,B 0,C 180,E1 -552.337,E2 -552.337} C_VEL
LIN {X 0,Y 601.364,Z 436.07,A -85,B 0,C 180,E1 -554.897,E2 -554.897} C_VEL
LIN {X 0,Y 601.358,Z 436.071,A -85,B 0,C 180,E1 -556.987,E2 -556.987} C_VEL
LIN {X 0,Y 601.374,Z 436.074,A -85,B 0,C 180,E1 -559.809,E2 -559.809} C_VEL
LIN {X 0,Y 601.385,Z 436.069,A -85,B 0,C 180,E1 -562.683,E2 -562.683} C_VEL
LIN {X 0,Y 601.358,Z 436.071,A -85,B 0,C 180,E1 -564.879,E2 -564.879} C_VEL
LIN {X 0,Y 601.373,Z 436.076,A -85,B 0,C 180,E1 -567.868,E2 -567.868} C_VEL
LIN {X 0,Y 601.392,Z 436.076,A -85,B 0,C 180,E1 -570.164,E2 -570.164} C_VEL
LIN {X 0,Y 601.38,Z 436.069,A -85,B 0,C 180,E1 -572.71,E2 -572.71} C_VEL
LIN {X 0,Y 601.343,Z 436.072,A -85,B 0,C 180,E1 -575.106,E2 -575.106} C_VEL
LIN {X 0,Y 601.375,Z 436.07,A -85,B 0,C 180,E1 -577.422,E2 -577.422} C_VEL
LIN {X 0,Y 601.38,Z 436.078,A -85,B 0,C 180,E1 -579.996,E2 -579.996} C_VEL
LIN {X 0,Y 601.348,Z 436.074,A -85,B 0,C 180,E1 -582.674,E2 -582.674} C_VEL
LIN {X 0,Y 601.384,Z 436.07,A -85,B 0,C 180,E1 -585.479,E2 -585.479} C_VEL
LIN {X 0,Y 601.388,Z 436.07,A -85,B 0,C 180,E1 -588.408,E2 -588.408} C_VEL
LIN {X 0,Y 601.361,Z 436.071,A -85,B 0,C 180,E1 -590.87,E2 -590.87} C_VEL
LIN {X 0,Y 601.372,Z 436.075,A -85,B 0,C 180,E1 -593.741,E2 -593.741} C_VEL
LIN {X 0,Y 601.365,Z 436.071,A -85,B 0,C 180,E1 -596.683,E2 -596.683} C_VEL
LIN {X 0,Y 601.37,Z 436.069,A -85,B 0,C 180,E1 -599.056,E2 -599.056} C_VEL
LIN {X 0,Y 601.355,Z 436.072,A -85,B 0,C 180,E1 -601.37,E2 -601.37} C_VEL
LIN {X 0,Y 601.38,Z 436.073,A -85,B 0,C 180,E1 -604.38,E2 -604.38} C_VEL
LIN {X 0,Y 601.359,Z 436.073,A -85,B 0,C 180,E1 -606.587,E2 -606.587} C_VEL
LIN {X 0,Y 601.388,Z 436.07,A -85,B 0,C 180,E1 -609.477,E2 -609.477} C_VEL
LIN {X 0,Y 601.36,Z 436.076,A -85,B 0,C 180,E1 -612.311,E2 -612.311} C_VEL
LIN {X 0,Y 601.371,Z 436.074,A -85,B 0,C 180,E1 -614.408,E2 -614.408} C_VEL
LIN {X 0,Y 601.374,Z 436.072,A -85,B 0,C 180,E1 -616.483,E2 -616.483} C_VEL
LIN {X 0,Y 601.345,Z 436.073,A -85,B 0,C 180,E1 -619.223,E2 -619.223} C_VEL
LIN {X 0,Y 601.417,Z 436.074,A -85,B 0,C 180,E1 -621.939,E2 -621.939} C_VEL
LIN {X 0,Y 601.372,Z 436.071,A -85,B 0,C 180,E1 -624.635,E2 -624.635} C_VEL
LIN {X 0,Y 601.383,Z 436.069,A -85,B 0,C 180,E1 -627.321,E2 -627.321} C_VEL
LIN {X 0,Y 601.43,Z 436.073,A -85,B 0,C 180,E1 -630,E2 -630} C_VEL
LIN {X 0,Y 601.383,Z 436.069,A -85,B 0,C 180,E1 -632.679,E2 -632.679} C_VEL
LIN {X 0,Y 601.372,Z 436.071,A -85,B 0,C 180,E1 -635.365,E2 -635.365} C_VEL
LIN {X 0,Y 601.417,Z 436.074,A -85,B 0,C 180,E1 -638.061,E2 -638.061} C_VEL
LIN {X 0,Y 601.361,Z 436.071,A -85,B 0,C 180,E1 -640.99,E2 -640.99} C_VEL
LIN {X 0,Y 601.374,Z 436.072,A -85,B 0,C 180,E1 -643.517,E2 -643.517} C_VEL
LIN {X 0,Y 601.395,Z 436.072,A -85,B 0,C 180,E1 -646.288,E2 -646.288} C_VEL
LIN {X 0,Y 601.38,Z 436.069,A -85,B 0,C 180,E1 -649.1,E2 -649.1} C_VEL
LIN {X 0,Y 601.364,Z 436.071,A -85,B 0,C 180,E1 -651.241,E2 -651.241} C_VEL
LIN {X 0,Y 601.422,Z 436.071,A -85,B 0,C 180,E1 -654.142,E2 -654.142} C_VEL
LIN {X 0,Y 601.356,Z 436.071,A -85,B 0,C 180,E1 -657.115,E2 -657.115} C_VEL
LIN {X 0,Y 601.39,Z 436.075,A -85,B 0,C 180,E1 -660.145,E2 -660.145} C_VEL
LIN {X 0,Y 601.376,Z 436.069,A -85,B 0,C 180,E1 -662.712,E2 -662.712} C_VEL
LIN {X 0,Y 601.341,Z 436.072,A -85,B 0,C 180,E1 -665.107,E2 -665.107} C_VEL
LIN {X 0,Y 601.374,Z 436.071,A -85,B 0,C 180,E1 -667.423,E2 -667.423} C_VEL
LIN {X 0,Y 601.38,Z 436.078,A -85,B 0,C 180,E1 -669.997,E2 -669.997} C_VEL
LIN {X 0,Y 601.345,Z 436.072,A -85,B 0,C 180,E1 -672.676,E2 -672.676} C_VEL
LIN {X 0,Y 601.384,Z 436.07,A -85,B 0,C 180,E1 -675.48,E2 -675.48} C_VEL
LIN {X 0,Y 601.389,Z 436.07,A -85,B 0,C 180,E1 -678.41,E2 -678.41} C_VEL
LIN {X 0,Y 601.361,Z 436.07,A -85,B 0,C 180,E1 -680.872,E2 -680.872} C_VEL
LIN {X 0,Y 601.374,Z 436.076,A -85,B 0,C 180,E1 -683.742,E2 -683.742} C_VEL
LIN {X 0,Y 601.368,Z 436.07,A -85,B 0,C 180,E1 -686.684,E2 -686.684} C_VEL
LIN {X 0,Y 601.373,Z 436.069,A -85,B 0,C 180,E1 -689.057,E2 -689.057} C_VEL
LIN {X 0,Y 601.36,Z 436.072,A -85,B 0,C 180,E1 -691.371,E2 -691.371} C_VEL
LIN {X 0,Y 601.38,Z 436.072,A -85,B 0,C 180,E1 -694.382,E2 -694.382} C_VEL
LIN {X 0,Y 601.362,Z 436.072,A -85,B 0,C 180,E1 -696.589,E2 -696.589} C_VEL
LIN {X 0,Y 601.394,Z 436.069,A -85,B 0,C 180,E1 -699.478,E2 -699.478} C_VEL
LIN {X 0,Y 601.362,Z 436.074,A -85,B 0,C 180,E1 -702.312,E2 -702.312} C_VEL
LIN {X 0,Y 601.374,Z 436.072,A -85,B 0,C 180,E1 -704.409,E2 -704.409} C_VEL
LIN {X 0,Y 601.379,Z 436.07,A -85,B 0,C 180,E1 -706.484,E2 -706.484} C_VEL
LIN {X 0,Y 601.351,Z 436.072,A -85,B 0,C 180,E1 -709.224,E2 -709.224} C_VEL
LIN {X 0,Y 601.423,Z 436.073,A -85,B 0,C 180,E1 -711.94,E2 -711.94} C_VEL
LIN {X 0,Y 601.376,Z 436.07,A -85,B 0,C 180,E1 -714.637,E2 -714.637} C_VEL
LIN {X 0,Y 601.392,Z 436.068,A -85,B 0,C 180,E1 -717.322,E2 -717.322} C_VEL
LIN {X 0,Y 601.438,Z 436.07,A -85,B 0,C 180,E1 -720.001,E2 -720.001} C_VEL
LIN {X 0,Y 601.389,Z 436.068,A -85,B 0,C 180,E1 -722.68,E2 -722.68} C_VEL
LIN {X 0,Y 601.381,Z 436.07,A -85,B 0,C 180,E1 -725.365,E2 -725.365} C_VEL
LIN {X 0,Y 601.426,Z 436.07,A -85,B 0,C 180,E1 -728.062,E2 -728.062} C_VEL
LIN {X 0,Y 601.369,Z 436.069,A -85,B 0,C 180,E1 -730.988,E2 -730.988} C_VEL
LIN {X 0,Y 601.384,Z 436.071,A -85,B 0,C 180,E1 -733.517,E2 -733.517} C_VEL
LIN {X 0,Y 601.399,Z 436.07,A -85,B 0,C 180,E1 -736.289,E2 -736.289} C_VEL
LIN {X 0,Y 601.359,Z 436.07,A -85,B 0,C 180,E1 -739.102,E2 -739.102} C_VEL
LIN {X 0,Y 601.373,Z 436.07,A -85,B 0,C 180,E1 -741.241,E2 -741.241} C_VEL
LIN {X 0,Y 601.426,Z 436.069,A -85,B 0,C 180,E1 -744.142,E2 -744.142} C_VEL
LIN {X 0,Y 601.365,Z 436.07,A -85,B 0,C 180,E1 -747.116,E2 -747.116} C_VEL
LIN {X 0,Y 601.401,Z 436.072,A -85,B 0,C 180,E1 -750.166,E2 -750.166} C_VEL
LIN {X 0,Y 601.383,Z 436.068,A -85,B 0,C 180,E1 -752.711,E2 -752.711} C_VEL
LIN {X 0,Y 601.348,Z 436.072,A -85,B 0,C 180,E1 -755.106,E2 -755.106} C_VEL
LIN {X 0,Y 601.385,Z 436.071,A -85,B 0,C 180,E1 -757.423,E2 -757.423} C_VEL
LIN {X 0,Y 601.394,Z 436.075,A -85,B 0,C 180,E1 -759.997,E2 -759.997} C_VEL
LIN {X 0,Y 601.35,Z 436.072,A -85,B 0,C 180,E1 -762.676,E2 -762.676} C_VEL
LIN {X 0,Y 601.399,Z 436.07,A -85,B 0,C 180,E1 -765.48,E2 -765.48} C_VEL
LIN {X 0,Y 601.398,Z 436.068,A -85,B 0,C 180,E1 -768.41,E2 -768.41} C_VEL
LIN {X 0,Y 601.37,Z 436.069,A -85,B 0,C 180,E1 -770.871,E2 -770.871} C_VEL
LIN {X 0,Y 601.385,Z 436.076,A -85,B 0,C 180,E1 -773.742,E2 -773.742} C_VEL
LIN {X 0,Y 601.38,Z 436.068,A -85,B 0,C 180,E1 -776.684,E2 -776.684} C_VEL
LIN {X 0,Y 601.374,Z 436.069,A -85,B 0,C 180,E1 -779.056,E2 -779.056} C_VEL
LIN {X 0,Y 601.369,Z 436.073,A -85,B 0,C 180,E1 -781.37,E2 -781.37} C_VEL
LIN {X 0,Y 601.385,Z 436.074,A -85,B 0,C 180,E1 -784.381,E2 -784.381} C_VEL
LIN {X 0,Y 601.455,Z 436.248,A -85,B 0,C 180,E1 -785.704,E2 -785.704} C_VEL
LIN {X 0,Y 601.571,Z 445.532,A -85,B 0,C 180,E1 -787.36,E2 -787.36} C_VEL
LIN {X 0,Y 601.527,Z 460.846,A -85,B 0,C 180,E1 -790.017,E2 -790.017} C_VEL
LIN {X 0,Y 601.492,Z 476.368,A -85,B 0,C 180,E1 -792.666,E2 -792.666} C_VEL
LIN {X 0,Y 601.454,Z 493.959,A -85,B 0,C 180,E1 -795.623,E2 -795.623} C_VEL
LIN {X 0,Y 601.447,Z 501.245,A -85,B 0,C 180,E1 -796.808,E2 -796.808} C_VEL
LIN {X 0,Y 601.646,Z 503.732,A -85,B 0,C 180,E1 -796.876,E2 -796.876} C_VEL
LIN {X 0,Y 601.616,Z 607.908,A -85,B 0,C 180,E1 -798.14,E2 -798.14} C_VEL
LIN {X 0,Y 601.591,Z 621.233,A -85,B 0,C 180,E1 -798.438,E2 -798.438} C_VEL
LIN {X 0,Y 601.547,Z 633.665,A -85,B 0,C 180,E1 -798.854,E2 -798.854} C_VEL
LIN {X 0,Y 601.521,Z 645.615,A -85,B 0,C 180,E1 -799.396,E2 -799.396} C_VEL
LIN {X 0,Y 601.484,Z 657.192,A -85,B 0,C 180,E1 -800.076,E2 -800.076} C_VEL
LIN {X 0,Y 601.444,Z 667.592,A -85,B 0,C 180,E1 -800.839,E2 -800.839} C_VEL
LIN {X 0,Y 601.429,Z 676.112,A -85,B 0,C 180,E1 -801.601,E2 -801.601} C_VEL
LIN {X 0,Y 601.418,Z 683.961,A -85,B 0,C 180,E1 -802.446,E2 -802.446} C_VEL
LIN {X 0,Y 601.37,Z 691.223,A -85,B 0,C 180,E1 -803.398,E2 -803.398} C_VEL
LIN {X 0,Y 601.372,Z 696.862,A -85,B 0,C 180,E1 -804.299,E2 -804.299} C_VEL
LIN {X 0,Y 601.336,Z 701.943,A -85,B 0,C 180,E1 -805.307,E2 -805.307} C_VEL
LIN {X 0,Y 601.368,Z 705.888,A -85,B 0,C 180,E1 -806.315,E2 -806.315} C_VEL
LIN {X 0,Y 601.325,Z 708.805,A -85,B 0,C 180,E1 -807.32,E2 -807.32} C_VEL
LIN {X 0,Y 601.343,Z 710.203,A -85,B 0,C 180,E1 -807.991,E2 -807.991} C_VEL
LIN {X 0,Y 601.339,Z 711.784,A -85,B 0,C 180,E1 -809.33,E2 -809.33} C_VEL
LIN {X 0,Y 601.335,Z 712,A -85,B 0,C 180,E1 -810,E2 -810} C_VEL
LIN {X 0,Y 601.347,Z 711.183,A -85,B 0,C 180,E1 -811.339,E2 -811.339} C_VEL
LIN {X 0,Y 601.343,Z 710.203,A -85,B 0,C 180,E1 -812.009,E2 -812.009} C_VEL
LIN {X 0,Y 601.325,Z 708.805,A -85,B 0,C 180,E1 -812.68,E2 -812.68} C_VEL
LIN {X 0,Y 601.368,Z 705.888,A -85,B 0,C 180,E1 -813.685,E2 -813.685} C_VEL
LIN {X 0,Y 601.336,Z 701.943,A -85,B 0,C 180,E1 -814.693,E2 -814.693} C_VEL
LIN {X 0,Y 601.372,Z 696.862,A -85,B 0,C 180,E1 -815.701,E2 -815.701} C_VEL
LIN {X 0,Y 601.382,Z 690.473,A -85,B 0,C 180,E1 -816.711,E2 -816.711} C_VEL
LIN {X 0,Y 601.396,Z 682.478,A -85,B 0,C 180,E1 -817.723,E2 -817.723} C_VEL
LIN {X 0,Y 601.423,Z 674.336,A -85,B 0,C 180,E1 -818.568,E2 -818.568} C_VEL
LIN {X 0,Y 601.453,Z 664.385,A -85,B 0,C 180,E1 -819.415,E2 -819.415} C_VEL
LIN {X 0,Y 601.502,Z 653.175,A -85,B 0,C 180,E1 -820.179,E2 -820.179} C_VEL
LIN {X 0,Y 601.538,Z 640.909,A -85,B 0,C 180,E1 -820.836,E2 -820.836} C_VEL
LIN {X 0,Y 601.566,Z 628.358,A -85,B 0,C 180,E1 -821.34,E2 -821.34} C_VEL
LIN {X 0,Y 601.607,Z 615.349,A -85,B 0,C 180,E1 -821.711,E2 -821.711} C_VEL
LIN {X 0,Y 601.626,Z 602.094,A -85,B 0,C 180,E1 -821.946,E2 -821.946} C_VEL
LIN {X 0,Y 601.536,Z 502.239,A -85,B 0,C 180,E1 -823.148,E2 -823.148} C_VEL
LIN {X 0,Y 601.428,Z 501.029,A -85,B 0,C 180,E1 -823.214,E2 -823.214} C_VEL
LIN {X 0,Y 601.464,Z 484.646,A -85,B 0,C 180,E1 -825.938,E2 -825.938} C_VEL
LIN {X 0,Y 601.526,Z 467.464,A -85,B 0,C 180,E1 -828.848,E2 -828.848} C_VEL
LIN {X 0,Y 601.572,Z 450.498,A -85,B 0,C 180,E1 -831.773,E2 -831.773} C_VEL
LIN {X 0,Y 601.55,Z 437.046,A -85,B 0,C 180,E1 -834.136,E2 -834.136} C_VEL
LIN {X 0,Y 601.413,Z 436.126,A -85,B 0,C 180,E1 -834.382,E2 -834.382} C_VEL
LIN {X 0,Y 601.364,Z 436.071,A -85,B 0,C 180,E1 -837.352,E2 -837.352} C_VEL
LIN {X 0,Y 601.404,Z 436.076,A -85,B 0,C 180,E1 -840.165,E2 -840.165} C_VEL
LIN {X 0,Y 601.39,Z 436.069,A -85,B 0,C 180,E1 -842.71,E2 -842.71} C_VEL
LIN {X 0,Y 601.35,Z 436.072,A -85,B 0,C 180,E1 -845.105,E2 -845.105} C_VEL
LIN {X 0,Y 601.382,Z 436.069,A -85,B 0,C 180,E1 -847.422,E2 -847.422} C_VEL
LIN {X 0,Y 601.393,Z 436.075,A -85,B 0,C 180,E1 -849.996,E2 -849.996} C_VEL
LIN {X 0,Y 601.356,Z 436.073,A -85,B 0,C 180,E1 -852.675,E2 -852.675} C_VEL
LIN {X 0,Y 601.369,Z 436.071,A -85,B 0,C 180,E1 -855.476,E2 -855.476} C_VEL
LIN {X 0,Y 601.397,Z 436.071,A -85,B 0,C 180,E1 -858.409,E2 -858.409} C_VEL
LIN {X 0,Y 601.37,Z 436.07,A -85,B 0,C 180,E1 -860.87,E2 -860.87} C_VEL
LIN {X 0,Y 601.383,Z 436.072,A -85,B 0,C 180,E1 -863.741,E2 -863.741} C_VEL
LIN {X 0,Y 601.377,Z 436.07,A -85,B 0,C 180,E1 -866.683,E2 -866.683} C_VEL
LIN {X 0,Y 601.378,Z 436.068,A -85,B 0,C 180,E1 -869.055,E2 -869.055} C_VEL
LIN {X 0,Y 601.36,Z 436.071,A -85,B 0,C 180,E1 -871.369,E2 -871.369} C_VEL
LIN {X 0,Y 601.391,Z 436.072,A -85,B 0,C 180,E1 -874.38,E2 -874.38} C_VEL
LIN {X 0,Y 601.366,Z 436.073,A -85,B 0,C 180,E1 -876.587,E2 -876.587} C_VEL
LIN {X 0,Y 601.394,Z 436.068,A -85,B 0,C 180,E1 -879.476,E2 -879.476} C_VEL
LIN {X 0,Y 601.369,Z 436.076,A -85,B 0,C 180,E1 -882.31,E2 -882.31} C_VEL
LIN {X 0,Y 601.378,Z 436.073,A -85,B 0,C 180,E1 -884.407,E2 -884.407} C_VEL
LIN {X 0,Y 601.384,Z 436.071,A -85,B 0,C 180,E1 -886.483,E2 -886.483} C_VEL
LIN {X 0,Y 601.35,Z 436.071,A -85,B 0,C 180,E1 -889.222,E2 -889.222} C_VEL
LIN {X 0,Y 601.426,Z 436.07,A -85,B 0,C 180,E1 -891.938,E2 -891.938} C_VEL
LIN {X 0,Y 601.381,Z 436.07,A -85,B 0,C 180,E1 -894.635,E2 -894.635} C_VEL
LIN {X 0,Y 601.389,Z 436.068,A -85,B 0,C 180,E1 -897.32,E2 -897.32} C_VEL
LIN {X 0,Y 601.438,Z 436.07,A -85,B 0,C 180,E1 -899.999,E2 -899.999} C_VEL
LIN {X 0,Y 601.392,Z 436.068,A -85,B 0,C 180,E1 -902.678,E2 -902.678} C_VEL
LIN {X 0,Y 601.377,Z 436.07,A -85,B 0,C 180,E1 -905.363,E2 -905.363} C_VEL
LIN {X 0,Y 601.423,Z 436.073,A -85,B 0,C 180,E1 -908.06,E2 -908.06} C_VEL
LIN {X 0,Y 601.351,Z 436.072,A -85,B 0,C 180,E1 -910.776,E2 -910.776} C_VEL
LIN {X 0,Y 601.37,Z 436.075,A -85,B 0,C 180,E1 -912.337,E2 -912.337} C_VEL
LIN {X 0,Y 600.678,Z 436.158,A -85,B 0,C 180,E1 -912.897,E2 -912.897} C_VEL
LIN {X 0,Y 597.82,Z 436.518,A -85,B 0,C 180,E1 -913.805,E2 -913.805} C_VEL
LIN {X 0,Y 595.423,Z 436.813,A -85,B 0,C 180,E1 -914.535,E2 -914.535} C_VEL
LIN {X 0,Y 594.397,Z 436.938,A -85,B 0,C 180,E1 -915.099,E2 -915.099} C_VEL
LIN {X 0,Y 594.313,Z 436.949,A -85,B 0,C 180,E1 -915.29,E2 -915.29} C_VEL
LIN {X 0,Y 594.317,Z 436.956,A -85,B 0,C 180,E1 -917.905,E2 -917.905} C_VEL
LIN {X 0,Y 594.34,Z 436.945,A -85,B 0,C 180,E1 -920.908,E2 -920.908} C_VEL
LIN {X 0,Y 594.348,Z 436.949,A -85,B 0,C 180,E1 -923.704,E2 -923.704} C_VEL
LIN {X 0,Y 594.325,Z 436.947,A -85,B 0,C 180,E1 -926.701,E2 -926.701} C_VEL
LIN {X 0,Y 594.322,Z 436.947,A -85,B 0,C 180,E1 -929,E2 -929} C_VEL
LIN {X 0,Y 594.353,Z 436.948,A -85,B 0,C 180,E1 -931.64,E2 -931.64} C_VEL
LIN {X 0,Y 594.336,Z 436.947,A -85,B 0,C 180,E1 -934.581,E2 -934.581} C_VEL
LIN {X 0,Y 594.343,Z 436.948,A -85,B 0,C 180,E1 -937.603,E2 -937.603} C_VEL
LIN {X 0,Y 594.339,Z 436.947,A -85,B 0,C 180,E1 -940.567,E2 -940.567} C_VEL
LIN {X 0,Y 594.323,Z 436.948,A -85,B 0,C 180,E1 -943.301,E2 -943.301} C_VEL
LIN {X 0,Y 594.328,Z 436.953,A -85,B 0,C 180,E1 -946.162,E2 -946.162} C_VEL
LIN {X 0,Y 594.342,Z 436.946,A -85,B 0,C 180,E1 -948.533,E2 -948.533} C_VEL
LIN {X 0,Y 594.345,Z 436.945,A -85,B 0,C 180,E1 -951.298,E2 -951.298} C_VEL
LIN {X 0,Y 594.326,Z 436.953,A -85,B 0,C 180,E1 -953.754,E2 -953.754} C_VEL
LIN {X 0,Y 594.335,Z 436.953,A -85,B 0,C 180,E1 -956.236,E2 -956.236} C_VEL
LIN {X 0,Y 594.338,Z 436.947,A -85,B 0,C 180,E1 -958.648,E2 -958.648} C_VEL
LIN {X 0,Y 594.318,Z 436.947,A -85,B 0,C 180,E1 -961.05,E2 -961.05} C_VEL
LIN {X 0,Y 594.349,Z 436.955,A -85,B 0,C 180,E1 -963.981,E2 -963.981} C_VEL
LIN {X 0,Y 594.342,Z 436.951,A -85,B 0,C 180,E1 -966.294,E2 -966.294} C_VEL
LIN {X 0,Y 594.359,Z 436.944,A -85,B 0,C 180,E1 -969.223,E2 -969.223} C_VEL
LIN {X 0,Y 594.314,Z 436.958,A -85,B 0,C 180,E1 -972.094,E2 -972.094} C_VEL
LIN {X 0,Y 594.324,Z 436.955,A -85,B 0,C 180,E1 -974.218,E2 -974.218} C_VEL
LIN {X 0,Y 594.346,Z 436.95,A -85,B 0,C 180,E1 -976.32,E2 -976.32} C_VEL
LIN {X 0,Y 594.325,Z 436.948,A -85,B 0,C 180,E1 -979.094,E2 -979.094} C_VEL
LIN {X 0,Y 594.359,Z 436.951,A -85,B 0,C 180,E1 -981.843,E2 -981.843} C_VEL
LIN {X 0,Y 594.342,Z 436.948,A -85,B 0,C 180,E1 -984.572,E2 -984.572} C_VEL
LIN {X 0,Y 594.35,Z 436.945,A -85,B 0,C 180,E1 -987.289,E2 -987.289} C_VEL
LIN {X 0,Y 594.398,Z 436.949,A -85,B 0,C 180,E1 -990,E2 -990} C_VEL
LIN {X 0,Y 594.35,Z 436.945,A -85,B 0,C 180,E1 -992.711,E2 -992.711} C_VEL
LIN {X 0,Y 594.342,Z 436.948,A -85,B 0,C 180,E1 -995.428,E2 -995.428} C_VEL
LIN {X 0,Y 594.359,Z 436.951,A -85,B 0,C 180,E1 -998.157,E2 -998.157} C_VEL
LIN {X 0,Y 594.327,Z 436.947,A -85,B 0,C 180,E1 -1001.052,E2 -1001.052} C_VEL
LIN {X 0,Y 594.346,Z 436.95,A -85,B 0,C 180,E1 -1003.68,E2 -1003.68} C_VEL
LIN {X 0,Y 594.315,Z 436.95,A -85,B 0,C 180,E1 -1006.7,E2 -1006.7} C_VEL
LIN {X 0,Y 594.334,Z 436.948,A -85,B 0,C 180,E1 -1009.335,E2 -1009.335} C_VEL
LIN {X 0,Y 594.326,Z 436.95,A -85,B 0,C 180,E1 -1011.505,E2 -1011.505} C_VEL
LIN {X 0,Y 594.349,Z 436.947,A -85,B 0,C 180,E1 -1014.448,E2 -1014.448} C_VEL
LIN {X 0,Y 594.322,Z 436.949,A -85,B 0,C 180,E1 -1016.702,E2 -1016.702} C_VEL
LIN {X 0,Y 594.318,Z 436.947,A -85,B 0,C 180,E1 -1019.002,E2 -1019.002} C_VEL
LIN {X 0,Y 594.35,Z 436.949,A -85,B 0,C 180,E1 -1021.642,E2 -1021.642} C_VEL
LIN {X 0,Y 594.334,Z 436.946,A -85,B 0,C 180,E1 -1024.583,E2 -1024.583} C_VEL
LIN {X 0,Y 594.341,Z 436.95,A -85,B 0,C 180,E1 -1027.605,E2 -1027.605} C_VEL
LIN {X 0,Y 594.331,Z 436.954,A -85,B 0,C 180,E1 -1029.772,E2 -1029.772} C_VEL
LIN {X 0,Y 594.32,Z 436.95,A -85,B 0,C 180,E1 -1032.379,E2 -1032.379} C_VEL
LIN {X 0,Y 594.321,Z 436.948,A -85,B 0,C 180,E1 -1035.195,E2 -1035.195} C_VEL
LIN {X 0,Y 594.36,Z 436.949,A -85,B 0,C 180,E1 -1038.153,E2 -1038.153} C_VEL
LIN {X 0,Y 594.347,Z 436.945,A -85,B 0,C 180,E1 -1041.299,E2 -1041.299} C_VEL
LIN {X 0,Y 594.328,Z 436.954,A -85,B 0,C 180,E1 -1043.756,E2 -1043.756} C_VEL
LIN {X 0,Y 594.339,Z 436.951,A -85,B 0,C 180,E1 -1046.238,E2 -1046.238} C_VEL
LIN {X 0,Y 594.341,Z 436.946,A -85,B 0,C 180,E1 -1048.65,E2 -1048.65} C_VEL
LIN {X 0,Y 594.322,Z 436.947,A -85,B 0,C 180,E1 -1051.052,E2 -1051.052} C_VEL
LIN {X 0,Y 594.337,Z 436.956,A -85,B 0,C 180,E1 -1053.986,E2 -1053.986} C_VEL
LIN {X 0,Y 594.348,Z 436.949,A -85,B 0,C 180,E1 -1056.296,E2 -1056.296} C_VEL
LIN {X 0,Y 594.366,Z 436.942,A -85,B 0,C 180,E1 -1059.224,E2 -1059.224} C_VEL
LIN {X 0,Y 594.317,Z 436.956,A -85,B 0,C 180,E1 -1062.095,E2 -1062.095} C_VEL
LIN {X 0,Y 594.328,Z 436.953,A -85,B 0,C 180,E1 -1064.219,E2 -1064.219} C_VEL
LIN {X 0,Y 594.352,Z 436.948,A -85,B 0,C 180,E1 -1066.322,E2 -1066.322} C_VEL
LIN {X 0,Y 594.321,Z 436.946,A -85,B 0,C 180,E1 -1068.957,E2 -1068.957} C_VEL
LIN {X 0,Y 594.365,Z 436.95,A -85,B 0,C 180,E1 -1071.844,E2 -1071.844} C_VEL
LIN {X 0,Y 594.346,Z 436.946,A -85,B 0,C 180,E1 -1074.573,E2 -1074.573} C_VEL
LIN {X 0,Y 594.359,Z 436.944,A -85,B 0,C 180,E1 -1077.29,E2 -1077.29} C_VEL
LIN {X 0,Y 594.406,Z 436.945,A -85,B 0,C 180,E1 -1080.001,E2 -1080.001} C_VEL
LIN {X 0,Y 594.357,Z 436.943,A -85,B 0,C 180,E1 -1082.712,E2 -1082.712} C_VEL
LIN {X 0,Y 594.352,Z 436.947,A -85,B 0,C 180,E1 -1085.429,E2 -1085.429} C_VEL
LIN {X 0,Y 594.367,Z 436.946,A -85,B 0,C 180,E1 -1088.158,E2 -1088.158} C_VEL
LIN {X 0,Y 594.326,Z 436.946,A -85,B 0,C 180,E1 -1091.045,E2 -1091.045} C_VEL
LIN {X 0,Y 594.357,Z 436.949,A -85,B 0,C 180,E1 -1093.68,E2 -1093.68} C_VEL
LIN {X 0,Y 594.322,Z 436.947,A -85,B 0,C 180,E1 -1096.698,E2 -1096.698} C_VEL
LIN {X 0,Y 594.328,Z 436.947,A -85,B 0,C 180,E1 -1099.337,E2 -1099.337} C_VEL
LIN {X 0,Y 594.336,Z 436.949,A -85,B 0,C 180,E1 -1101.505,E2 -1101.505} C_VEL
LIN {X 0,Y 594.363,Z 436.944,A -85,B 0,C 180,E1 -1104.448,E2 -1104.448} C_VEL
LIN {X 0,Y 594.331,Z 436.945,A -85,B 0,C 180,E1 -1106.703,E2 -1106.703} C_VEL
LIN {X 0,Y 594.35,Z 436.952,A -85,B 0,C 180,E1 -1109.778,E2 -1109.778} C_VEL
LIN {X 0,Y 594.34,Z 436.951,A -85,B 0,C 180,E1 -1112.15,E2 -1112.15} C_VEL
LIN {X 0,Y 594.343,Z 436.945,A -85,B 0,C 180,E1 -1114.583,E2 -1114.583} C_VEL
LIN {X 0,Y 594.349,Z 436.95,A -85,B 0,C 180,E1 -1117.604,E2 -1117.604} C_VEL
LIN {X 0,Y 594.322,Z 436.948,A -85,B 0,C 180,E1 -1120.572,E2 -1120.572} C_VEL
LIN {X 0,Y 594.313,Z 436.949,A -85,B 0,C 180,E1 -1122.847,E2 -1122.847} C_VEL
LIN {X 0,Y 594.354,Z 436.952,A -85,B 0,C 180,E1 -1125.762,E2 -1125.762} C_VEL
LIN {X 0,Y 594.352,Z 436.944,A -85,B 0,C 180,E1 -1128.534,E2 -1128.534} C_VEL
LIN {X 0,Y 594.359,Z 436.945,A -85,B 0,C 180,E1 -1131.3,E2 -1131.3} C_VEL
LIN {X 0,Y 594.339,Z 436.954,A -85,B 0,C 180,E1 -1133.755,E2 -1133.755} C_VEL
LIN {X 0,Y 594.342,Z 436.949,A -85,B 0,C 180,E1 -1136.237,E2 -1136.237} C_VEL
LIN {X 0,Y 594.323,Z 436.948,A -85,B 0,C 180,E1 -1138.647,E2 -1138.647} C_VEL
LIN {X 0,Y 594.334,Z 436.947,A -85,B 0,C 180,E1 -1141.052,E2 -1141.052} C_VEL
LIN {X 0,Y 594.333,Z 436.956,A -85,B 0,C 180,E1 -1143.989,E2 -1143.989} C_VEL
LIN {X 0,Y 594.4,Z 437.163,A -85,B 0,C 180,E1 -1145.565,E2 -1145.565} C_VEL
LIN {X 0,Y 594.651,Z 442.22,A -85,B 0,C 180,E1 -1146.492,E2 -1146.492} C_VEL
LIN {X 0,Y 594.542,Z 457.742,A -85,B 0,C 180,E1 -1149.23,E2 -1149.23} C_VEL
LIN {X 0,Y 594.501,Z 473.263,A -85,B 0,C 180,E1 -1151.922,E2 -1151.922} C_VEL
LIN {X 0,Y 594.393,Z 490.855,A -85,B 0,C 180,E1 -1154.923,E2 -1154.923} C_VEL
LIN {X 0,Y 594.426,Z 501.239,A -85,B 0,C 180,E1 -1156.649,E2 -1156.649} C_VEL
LIN {X 0,Y 594.73,Z 503.732,A -85,B 0,C 180,E1 -1156.721,E2 -1156.721} C_VEL
LIN {X 0,Y 594.666,Z 607.857,A -85,B 0,C 180,E1 -1157.999,E2 -1157.999} C_VEL
LIN {X 0,Y 594.639,Z 621.24,A -85,B 0,C 180,E1 -1158.301,E2 -1158.301} C_VEL
LIN {X 0,Y 594.593,Z 634.353,A -85,B 0,C 180,E1 -1158.748,E2 -1158.748} C_VEL
LIN {X 0,Y 594.537,Z 645.601,A -85,B 0,C 180,E1 -1159.27,E2 -1159.27} C_VEL
LIN {X 0,Y 594.472,Z 657.188,A -85,B 0,C 180,E1 -1159.958,E2 -1159.958} C_VEL
LIN {X 0,Y 594.414,Z 667.591,A -85,B 0,C 180,E1 -1160.73,E2 -1160.73} C_VEL
LIN {X 0,Y 594.373,Z 677.79,A -85,B 0,C 180,E1 -1161.672,E2 -1161.672} C_VEL
LIN {X 0,Y 594.317,Z 686.689,A -85,B 0,C 180,E1 -1162.697,E2 -1162.697} C_VEL
LIN {X 0,Y 594.281,Z 693.163,A -85,B 0,C 180,E1 -1163.615,E2 -1163.615} C_VEL
LIN {X 0,Y 594.289,Z 698.671,A -85,B 0,C 180,E1 -1164.571,E2 -1164.571} C_VEL
LIN {X 0,Y 594.27,Z 703.358,A -85,B 0,C 180,E1 -1165.591,E2 -1165.591} C_VEL
LIN {X 0,Y 594.267,Z 706.948,A -85,B 0,C 180,E1 -1166.61,E2 -1166.61} C_VEL
LIN {X 0,Y 594.225,Z 708.799,A -85,B 0,C 180,E1 -1167.288,E2 -1167.288} C_VEL
LIN {X 0,Y 594.241,Z 710.204,A -85,B 0,C 180,E1 -1167.967,E2 -1167.967} C_VEL
LIN {X 0,Y 594.239,Z 711.785,A -85,B 0,C 180,E1 -1169.322,E2 -1169.322} C_VEL
LIN {X 0,Y 594.236,Z 712,A -85,B 0,C 180,E1 -1170,E2 -1170} C_VEL
LIN {X 0,Y 594.247,Z 711.183,A -85,B 0,C 180,E1 -1171.355,E2 -1171.355} C_VEL
LIN {X 0,Y 594.241,Z 710.204,A -85,B 0,C 180,E1 -1172.033,E2 -1172.033} C_VEL
LIN {X 0,Y 594.225,Z 708.799,A -85,B 0,C 180,E1 -1172.712,E2 -1172.712} C_VEL
LIN {X 0,Y 594.289,Z 705.882,A -85,B 0,C 180,E1 -1173.729,E2 -1173.729} C_VEL
LIN {X 0,Y 594.241,Z 701.937,A -85,B 0,C 180,E1 -1174.749,E2 -1174.749} C_VEL
LIN {X 0,Y 594.298,Z 696.859,A -85,B 0,C 180,E1 -1175.769,E2 -1175.769} C_VEL
LIN {X 0,Y 594.316,Z 690.474,A -85,B 0,C 180,E1 -1176.791,E2 -1176.791} C_VEL
LIN {X 0,Y 594.346,Z 682.479,A -85,B 0,C 180,E1 -1177.815,E2 -1177.815} C_VEL
LIN {X 0,Y 594.377,Z 674.336,A -85,B 0,C 180,E1 -1178.671,E2 -1178.671} C_VEL
LIN {X 0,Y 594.416,Z 664.373,A -85,B 0,C 180,E1 -1179.528,E2 -1179.528} C_VEL
LIN {X 0,Y 594.476,Z 653.179,A -85,B 0,C 180,E1 -1180.3,E2 -1180.3} C_VEL
LIN {X 0,Y 594.56,Z 640.712,A -85,B 0,C 180,E1 -1180.974,E2 -1180.974} C_VEL
LIN {X 0,Y 594.6,Z 628.658,A -85,B 0,C 180,E1 -1181.464,E2 -1181.464} C_VEL
LIN {X 0,Y 594.645,Z 616.258,A -85,B 0,C 180,E1 -1181.828,E2 -1181.828} C_VEL
LIN {X 0,Y 594.665,Z 603.61,A -85,B 0,C 180,E1 -1182.066,E2 -1182.066} C_VEL
LIN {X 0,Y 594.576,Z 502.67,A -85,B 0,C 180,E1 -1183.296,E2 -1183.296} C_VEL
LIN {X 0,Y 594.398,Z 501.028,A -85,B 0,C 180,E1 -1183.374,E2 -1183.374} C_VEL
LIN {X 0,Y 594.43,Z 484.646,A -85,B 0,C 180,E1 -1186.131,E2 -1186.131} C_VEL
LIN {X 0,Y 594.541,Z 468.695,A -85,B 0,C 180,E1 -1188.865,E2 -1188.865} C_VEL
LIN {X 0,Y 594.603,Z 451.533,A -85,B 0,C 180,E1 -1191.858,E2 -1191.858} C_VEL
LIN {X 0,Y 594.665,Z 439.144,A -85,B 0,C 180,E1 -1194.057,E2 -1194.057} C_VEL
LIN {X 0,Y 594.379,Z 437.02,A -85,B 0,C 180,E1 -1194.493,E2 -1194.493} C_VEL
LIN {X 0,Y 594.325,Z 436.95,A -85,B 0,C 180,E1 -1197.515,E2 -1197.515} C_VEL
LIN {X 0,Y 594.366,Z 436.949,A -85,B 0,C 180,E1 -1200.324,E2 -1200.324} C_VEL
LIN {X 0,Y 594.337,Z 436.946,A -85,B 0,C 180,E1 -1202.952,E2 -1202.952} C_VEL
LIN {X 0,Y 594.306,Z 436.951,A -85,B 0,C 180,E1 -1205.412,E2 -1205.412} C_VEL
LIN {X 0,Y 594.363,Z 436.95,A -85,B 0,C 180,E1 -1207.942,E2 -1207.942} C_VEL
LIN {X 0,Y 594.323,Z 436.947,A -85,B 0,C 180,E1 -1210.815,E2 -1210.815} C_VEL
LIN {X 0,Y 594.336,Z 436.946,A -85,B 0,C 180,E1 -1213.302,E2 -1213.302} C_VEL
LIN {X 0,Y 594.334,Z 436.956,A -85,B 0,C 180,E1 -1216.163,E2 -1216.163} C_VEL
LIN {X 0,Y 594.352,Z 436.947,A -85,B 0,C 180,E1 -1218.533,E2 -1218.533} C_VEL
LIN {X 0,Y 594.324,Z 436.947,A -85,B 0,C 180,E1 -1221.302,E2 -1221.302} C_VEL
LIN {X 0,Y 594.338,Z 436.95,A -85,B 0,C 180,E1 -1223.754,E2 -1223.754} C_VEL
LIN {X 0,Y 594.349,Z 436.952,A -85,B 0,C 180,E1 -1226.236,E2 -1226.236} C_VEL
LIN {X 0,Y 594.349,Z 436.946,A -85,B 0,C 180,E1 -1228.648,E2 -1228.648} C_VEL
LIN {X 0,Y 594.33,Z 436.946,A -85,B 0,C 180,E1 -1231.05,E2 -1231.05} C_VEL
LIN {X 0,Y 594.347,Z 436.952,A -85,B 0,C 180,E1 -1233.984,E2 -1233.984} C_VEL
LIN {X 0,Y 594.349,Z 436.951,A -85,B 0,C 180,E1 -1236.293,E2 -1236.293} C_VEL
LIN {X 0,Y 594.368,Z 436.941,A -85,B 0,C 180,E1 -1239.222,E2 -1239.222} C_VEL
LIN {X 0,Y 594.322,Z 436.956,A -85,B 0,C 180,E1 -1242.093,E2 -1242.093} C_VEL
LIN {X 0,Y 594.331,Z 436.954,A -85,B 0,C 180,E1 -1244.217,E2 -1244.217} C_VEL
LIN {X 0,Y 594.358,Z 436.949,A -85,B 0,C 180,E1 -1246.32,E2 -1246.32} C_VEL
LIN {X 0,Y 594.316,Z 436.947,A -85,B 0,C 180,E1 -1249.093,E2 -1249.093} C_VEL
LIN {X 0,Y 594.367,Z 436.946,A -85,B 0,C 180,E1 -1251.842,E2 -1251.842} C_VEL
LIN {X 0,Y 594.352,Z 436.947,A -85,B 0,C 180,E1 -1254.571,E2 -1254.571} C_VEL
LIN {X 0,Y 594.357,Z 436.943,A -85,B 0,C 180,E1 -1257.288,E2 -1257.288} C_VEL
LIN {X 0,Y 594.406,Z 436.945,A -85,B 0,C 180,E1 -1259.999,E2 -1259.999} C_VEL
LIN {X 0,Y 594.359,Z 436.944,A -85,B 0,C 180,E1 -1262.71,E2 -1262.71} C_VEL
LIN {X 0,Y 594.346,Z 436.946,A -85,B 0,C 180,E1 -1265.427,E2 -1265.427} C_VEL
LIN {X 0,Y 594.365,Z 436.95,A -85,B 0,C 180,E1 -1268.156,E2 -1268.156} C_VEL
LIN {X 0,Y 594.321,Z 436.946,A -85,B 0,C 180,E1 -1271.043,E2 -1271.043} C_VEL
LIN {X 0,Y 594.352,Z 436.948,A -85,B 0,C 180,E1 -1273.678,E2 -1273.678} C_VEL
LIN {X 0,Y 594.313,Z 436.949,A -85,B 0,C 180,E1 -1275.29,E2 -1275.29} C_VEL
LIN {X 0,Y 593.648,Z 437.04,A -85,B 0,C 180,E1 -1275.855,E2 -1275.855} C_VEL
LIN {X 0,Y 590.795,Z 437.399,A -85,B 0,C 180,E1 -1276.773,E2 -1276.773} C_VEL
LIN {X 0,Y 588.383,Z 437.7,A -85,B 0,C 180,E1 -1277.511,E2 -1277.511} C_VEL
LIN {X 0,Y 587.347,Z 437.824,A -85,B 0,C 180,E1 -1278.081,E2 -1278.081} C_VEL
LIN {X 0,Y 587.263,Z 437.831,A -85,B 0,C 180,E1 -1278.274,E2 -1278.274} C_VEL
LIN {X 0,Y 587.304,Z 437.821,A -85,B 0,C 180,E1 -1281.037,E2 -1281.037} C_VEL
LIN {X 0,Y 587.292,Z 437.833,A -85,B 0,C 180,E1 -1284.007,E2 -1284.007} C_VEL
LIN {X 0,Y 587.278,Z 437.83,A -85,B 0,C 180,E1 -1286.28,E2 -1286.28} C_VEL
LIN {X 0,Y 587.285,Z 437.823,A -85,B 0,C 180,E1 -1289.123,E2 -1289.123} C_VEL
LIN {X 0,Y 587.301,Z 437.829,A -85,B 0,C 180,E1 -1291.83,E2 -1291.83} C_VEL
LIN {X 0,Y 587.313,Z 437.825,A -85,B 0,C 180,E1 -1294.344,E2 -1294.344} C_VEL
LIN {X 0,Y 587.299,Z 437.826,A -85,B 0,C 180,E1 -1297.609,E2 -1297.609} C_VEL
LIN {X 0,Y 587.286,Z 437.83,A -85,B 0,C 180,E1 -1300.255,E2 -1300.255} C_VEL
LIN {X 0,Y 587.267,Z 437.826,A -85,B 0,C 180,E1 -1303.114,E2 -1303.114} C_VEL
LIN {X 0,Y 587.284,Z 437.832,A -85,B 0,C 180,E1 -1306.046,E2 -1306.046} C_VEL
LIN {X 0,Y 587.271,Z 437.824,A -85,B 0,C 180,E1 -1308.93,E2 -1308.93} C_VEL
LIN {X 0,Y 587.294,Z 437.825,A -85,B 0,C 180,E1 -1311.518,E2 -1311.518} C_VEL
LIN {X 0,Y 587.258,Z 437.835,A -85,B 0,C 180,E1 -1314.098,E2 -1314.098} C_VEL
LIN {X 0,Y 587.291,Z 437.825,A -85,B 0,C 180,E1 -1316.601,E2 -1316.601} C_VEL
LIN {X 0,Y 587.297,Z 437.823,A -85,B 0,C 180,E1 -1319.032,E2 -1319.032} C_VEL
LIN {X 0,Y 587.265,Z 437.827,A -85,B 0,C 180,E1 -1321.4,E2 -1321.4} C_VEL
LIN {X 0,Y 587.293,Z 437.831,A -85,B 0,C 180,E1 -1323.828,E2 -1323.828} C_VEL
LIN {X 0,Y 587.285,Z 437.825,A -85,B 0,C 180,E1 -1326.74,E2 -1326.74} C_VEL
LIN {X 0,Y 587.29,Z 437.829,A -85,B 0,C 180,E1 -1329.694,E2 -1329.694} C_VEL
LIN {X 0,Y 587.265,Z 437.835,A -85,B 0,C 180,E1 -1331.872,E2 -1331.872} C_VEL
LIN {X 0,Y 587.281,Z 437.826,A -85,B 0,C 180,E1 -1334.736,E2 -1334.736} C_VEL
LIN {X 0,Y 587.256,Z 437.828,A -85,B 0,C 180,E1 -1336.857,E2 -1336.857} C_VEL
LIN {X 0,Y 587.305,Z 437.827,A -85,B 0,C 180,E1 -1339.66,E2 -1339.66} C_VEL
LIN {X 0,Y 587.292,Z 437.828,A -85,B 0,C 180,E1 -1342.436,E2 -1342.436} C_VEL
LIN {X 0,Y 587.308,Z 437.822,A -85,B 0,C 180,E1 -1345.195,E2 -1345.195} C_VEL
LIN {X 0,Y 587.359,Z 437.825,A -85,B 0,C 180,E1 -1347.943,E2 -1347.943} C_VEL
LIN {X 0,Y 587.366,Z 437.825,A -85,B 0,C 180,E1 -1350,E2 -1350} C_VEL
LIN {X 0,Y 587.318,Z 437.821,A -85,B 0,C 180,E1 -1352.743,E2 -1352.743} C_VEL
LIN {X 0,Y 587.311,Z 437.824,A -85,B 0,C 180,E1 -1355.493,E2 -1355.493} C_VEL
LIN {X 0,Y 587.317,Z 437.827,A -85,B 0,C 180,E1 -1358.256,E2 -1358.256} C_VEL
LIN {X 0,Y 587.297,Z 437.823,A -85,B 0,C 180,E1 -1361.117,E2 -1361.117} C_VEL
LIN {X 0,Y 587.33,Z 437.827,A -85,B 0,C 180,E1 -1363.846,E2 -1363.846} C_VEL
LIN {X 0,Y 587.267,Z 437.827,A -85,B 0,C 180,E1 -1366.794,E2 -1366.794} C_VEL
LIN {X 0,Y 587.28,Z 437.829,A -85,B 0,C 180,E1 -1369.577,E2 -1369.577} C_VEL
LIN {X 0,Y 587.285,Z 437.832,A -85,B 0,C 180,E1 -1371.775,E2 -1371.775} C_VEL
LIN {X 0,Y 587.291,Z 437.826,A -85,B 0,C 180,E1 -1374.571,E2 -1374.571} C_VEL
LIN {X 0,Y 587.272,Z 437.826,A -85,B 0,C 180,E1 -1377.049,E2 -1377.049} C_VEL
LIN {X 0,Y 587.297,Z 437.83,A -85,B 0,C 180,E1 -1380.172,E2 -1380.172} C_VEL
LIN {X 0,Y 587.293,Z 437.824,A -85,B 0,C 180,E1 -1382.581,E2 -1382.581} C_VEL
LIN {X 0,Y 587.275,Z 437.823,A -85,B 0,C 180,E1 -1385.059,E2 -1385.059} C_VEL
LIN {X 0,Y 587.301,Z 437.83,A -85,B 0,C 180,E1 -1387.836,E2 -1387.836} C_VEL
LIN {X 0,Y 587.272,Z 437.829,A -85,B 0,C 180,E1 -1390.257,E2 -1390.257} C_VEL
LIN {X 0,Y 587.266,Z 437.824,A -85,B 0,C 180,E1 -1393.115,E2 -1393.115} C_VEL
LIN {X 0,Y 587.284,Z 437.834,A -85,B 0,C 180,E1 -1396.048,E2 -1396.048} C_VEL
LIN {X 0,Y 587.287,Z 437.823,A -85,B 0,C 180,E1 -1398.93,E2 -1398.93} C_VEL
LIN {X 0,Y 587.297,Z 437.826,A -85,B 0,C 180,E1 -1401.52,E2 -1401.52} C_VEL
LIN {X 0,Y 587.26,Z 437.834,A -85,B 0,C 180,E1 -1404.1,E2 -1404.1} C_VEL
LIN {X 0,Y 587.295,Z 437.824,A -85,B 0,C 180,E1 -1406.603,E2 -1406.603} C_VEL
LIN {X 0,Y 587.3,Z 437.822,A -85,B 0,C 180,E1 -1409.033,E2 -1409.033} C_VEL
LIN {X 0,Y 587.269,Z 437.828,A -85,B 0,C 180,E1 -1411.402,E2 -1411.402} C_VEL
LIN {X 0,Y 587.289,Z 437.83,A -85,B 0,C 180,E1 -1413.832,E2 -1413.832} C_VEL
LIN {X 0,Y 587.291,Z 437.824,A -85,B 0,C 180,E1 -1416.741,E2 -1416.741} C_VEL
LIN {X 0,Y 587.296,Z 437.828,A -85,B 0,C 180,E1 -1419.695,E2 -1419.695} C_VEL
LIN {X 0,Y 587.261,Z 437.828,A -85,B 0,C 180,E1 -1422.593,E2 -1422.593} C_VEL
LIN {X 0,Y 587.304,Z 437.825,A -85,B 0,C 180,E1 -1425.447,E2 -1425.447} C_VEL
LIN {X 0,Y 587.307,Z 437.824,A -85,B 0,C 180,E1 -1428.264,E2 -1428.264} C_VEL
LIN {X 0,Y 587.269,Z 437.824,A -85,B 0,C 180,E1 -1431.051,E2 -1431.051} C_VEL
LIN {X 0,Y 587.3,Z 437.83,A -85,B 0,C 180,E1 -1433.818,E2 -1433.818} C_VEL
LIN {X 0,Y 587.298,Z 437.832,A -85,B 0,C 180,E1 -1435.884,E2 -1435.884} C_VEL
LIN {X 0,Y 587.363,Z 437.823,A -85,B 0,C 180,E1 -1437.944,E2 -1437.944} C_VEL
LIN {X 0,Y 587.374,Z 437.821,A -85,B 0,C 180,E1 -1440.001,E2 -1440.001} C_VEL
LIN {X 0,Y 587.325,Z 437.819,A -85,B 0,C 180,E1 -1442.744,E2 -1442.744} C_VEL
LIN {X 0,Y 587.321,Z 437.823,A -85,B 0,C 180,E1 -1445.494,E2 -1445.494} C_VEL
LIN {X 0,Y 587.322,Z 437.822,A -85,B 0,C 180,E1 -1448.257,E2 -1448.257} C_VEL
LIN {X 0,Y 587.292,Z 437.822,A -85,B 0,C 180,E1 -1451.108,E2 -1451.108} C_VEL
LIN {X 0,Y 587.336,Z 437.827,A -85,B 0,C 180,E1 -1453.847,E2 -1453.847} C_VEL
LIN {X 0,Y 587.275,Z 437.824,A -85,B 0,C 180,E1 -1456.792,E2 -1456.792} C_VEL
LIN {X 0,Y 587.28,Z 437.827,A -85,B 0,C 180,E1 -1459.578,E2 -1459.578} C_VEL
LIN {X 0,Y 587.298,Z 437.824,A -85,B 0,C 180,E1 -1462.516,E2 -1462.516} C_VEL
LIN {X 0,Y 587.297,Z 437.826,A -85,B 0,C 180,E1 -1465.519,E2 -1465.519} C_VEL
LIN {X 0,Y 587.282,Z 437.832,A -85,B 0,C 180,E1 -1467.822,E2 -1467.822} C_VEL
LIN {X 0,Y 587.312,Z 437.822,A -85,B 0,C 180,E1 -1470.507,E2 -1470.507} C_VEL
LIN {X 0,Y 587.282,Z 437.824,A -85,B 0,C 180,E1 -1473.104,E2 -1473.104} C_VEL
LIN {X 0,Y 587.258,Z 437.831,A -85,B 0,C 180,E1 -1475.533,E2 -1475.533} C_VEL
LIN {X 0,Y 587.303,Z 437.832,A -85,B 0,C 180,E1 -1477.835,E2 -1477.835} C_VEL
LIN {X 0,Y 587.284,Z 437.828,A -85,B 0,C 180,E1 -1480.258,E2 -1480.258} C_VEL
LIN {X 0,Y 587.276,Z 437.826,A -85,B 0,C 180,E1 -1483.115,E2 -1483.115} C_VEL
LIN {X 0,Y 587.298,Z 437.83,A -85,B 0,C 180,E1 -1486.048,E2 -1486.048} C_VEL
LIN {X 0,Y 587.281,Z 437.823,A -85,B 0,C 180,E1 -1488.932,E2 -1488.932} C_VEL
LIN {X 0,Y 587.308,Z 437.826,A -85,B 0,C 180,E1 -1491.519,E2 -1491.519} C_VEL
LIN {X 0,Y 587.258,Z 437.829,A -85,B 0,C 180,E1 -1494.468,E2 -1494.468} C_VEL
LIN {X 0,Y 587.284,Z 437.824,A -85,B 0,C 180,E1 -1496.897,E2 -1496.897} C_VEL
LIN {X 0,Y 587.313,Z 437.825,A -85,B 0,C 180,E1 -1499.495,E2 -1499.495} C_VEL
LIN {X 0,Y 587.286,Z 437.829,A -85,B 0,C 180,E1 -1502.32,E2 -1502.32} C_VEL
LIN {X 0,Y 587.353,Z 437.915,A -85,B 0,C 180,E1 -1505.372,E2 -1505.372} C_VEL
LIN {X 0,Y 587.738,Z 442.22,A -85,B 0,C 180,E1 -1506.199,E2 -1506.199} C_VEL
LIN {X 0,Y 587.574,Z 457.742,A -85,B 0,C 180,E1 -1508.972,E2 -1508.972} C_VEL
LIN {X 0,Y 587.484,Z 473.263,A -85,B 0,C 180,E1 -1511.698,E2 -1511.698} C_VEL
LIN {X 0,Y 587.369,Z 489.82,A -85,B 0,C 180,E1 -1514.56,E2 -1514.56} C_VEL
LIN {X 0,Y 587.394,Z 501.236,A -85,B 0,C 180,E1 -1516.486,E2 -1516.486} C_VEL
LIN {X 0,Y 587.73,Z 503.732,A -85,B 0,C 180,E1 -1516.56,E2 -1516.56} C_VEL
LIN {X 0,Y 587.728,Z 607.806,A -85,B 0,C 180,E1 -1517.855,E2 -1517.855} C_VEL
LIN {X 0,Y 587.679,Z 620.488,A -85,B 0,C 180,E1 -1518.139,E2 -1518.139} C_VEL
LIN {X 0,Y 587.611,Z 633.791,A -85,B 0,C 180,E1 -1518.59,E2 -1518.59} C_VEL
LIN {X 0,Y 587.555,Z 645.587,A -85,B 0,C 180,E1 -1519.141,E2 -1519.141} C_VEL
LIN {X 0,Y 587.456,Z 657.185,A -85,B 0,C 180,E1 -1519.836,E2 -1519.836} C_VEL
LIN {X 0,Y 587.393,Z 667.59,A -85,B 0,C 180,E1 -1520.618,E2 -1520.618} C_VEL
LIN {X 0,Y 587.33,Z 677.79,A -85,B 0,C 180,E1 -1521.571,E2 -1521.571} C_VEL
LIN {X 0,Y 587.259,Z 686.68,A -85,B 0,C 180,E1 -1522.608,E2 -1522.608} C_VEL
LIN {X 0,Y 587.194,Z 693.72,A -85,B 0,C 180,E1 -1523.628,E2 -1523.628} C_VEL
LIN {X 0,Y 587.211,Z 698.663,A -85,B 0,C 180,E1 -1524.506,E2 -1524.506} C_VEL
LIN {X 0,Y 587.189,Z 703.352,A -85,B 0,C 180,E1 -1525.538,E2 -1525.538} C_VEL
LIN {X 0,Y 587.193,Z 706.944,A -85,B 0,C 180,E1 -1526.569,E2 -1526.569} C_VEL
LIN {X 0,Y 587.132,Z 708.792,A -85,B 0,C 180,E1 -1527.256,E2 -1527.256} C_VEL
LIN {X 0,Y 587.14,Z 710.205,A -85,B 0,C 180,E1 -1527.942,E2 -1527.942} C_VEL
LIN {X 0,Y 587.14,Z 711.785,A -85,B 0,C 180,E1 -1529.314,E2 -1529.314} C_VEL
LIN {X 0,Y 587.137,Z 712,A -85,B 0,C 180,E1 -1530,E2 -1530} C_VEL
LIN {X 0,Y 587.147,Z 711.182,A -85,B 0,C 180,E1 -1531.372,E2 -1531.372} C_VEL
LIN {X 0,Y 587.14,Z 710.205,A -85,B 0,C 180,E1 -1532.058,E2 -1532.058} C_VEL
LIN {X 0,Y 587.132,Z 708.792,A -85,B 0,C 180,E1 -1532.744,E2 -1532.744} C_VEL
LIN {X 0,Y 587.213,Z 705.875,A -85,B 0,C 180,E1 -1533.774,E2 -1533.774} C_VEL
LIN {X 0,Y 587.146,Z 701.932,A -85,B 0,C 180,E1 -1534.806,E2 -1534.806} C_VEL
LIN {X 0,Y 587.229,Z 696.856,A -85,B 0,C 180,E1 -1535.839,E2 -1535.839} C_VEL
LIN {X 0,Y 587.245,Z 689.24,A -85,B 0,C 180,E1 -1537.046,E2 -1537.046} C_VEL
LIN {X 0,Y 587.3,Z 680.969,A -85,B 0,C 180,E1 -1538.083,E2 -1538.083} C_VEL
LIN {X 0,Y 587.343,Z 672.502,A -85,B 0,C 180,E1 -1538.949,E2 -1538.949} C_VEL
LIN {X 0,Y 587.419,Z 662.1,A -85,B 0,C 180,E1 -1539.816,E2 -1539.816} C_VEL
LIN {X 0,Y 587.529,Z 650.312,A -85,B 0,C 180,E1 -1540.598,E2 -1540.598} C_VEL
LIN {X 0,Y 587.568,Z 638.311,A -85,B 0,C 180,E1 -1541.213,E2 -1541.213} C_VEL
LIN {X 0,Y 587.651,Z 626.213,A -85,B 0,C 180,E1 -1541.684,E2 -1541.684} C_VEL
LIN {X 0,Y 587.737,Z 613.51,A -85,B 0,C 180,E1 -1542.035,E2 -1542.035} C_VEL
LIN {X 0,Y 587.787,Z 598.532,A -85,B 0,C 180,E1 -1542.275,E2 -1542.275} C_VEL
LIN {X 0,Y 587.73,Z 503.732,A -85,B 0,C 180,E1 -1543.44,E2 -1543.44} C_VEL
LIN {X 0,Y 587.394,Z 501.237,A -85,B 0,C 180,E1 -1543.514,E2 -1543.514} C_VEL
LIN {X 0,Y 587.427,Z 485.681,A -85,B 0,C 180,E1 -1546.15,E2 -1546.15} C_VEL
LIN {X 0,Y 587.54,Z 470.159,A -85,B 0,C 180,E1 -1548.842,E2 -1548.842} C_VEL
LIN {X 0,Y 587.634,Z 453.602,A -85,B 0,C 180,E1 -1551.762,E2 -1551.762} C_VEL
LIN {X 0,Y 587.751,Z 441.185,A -85,B 0,C 180,E1 -1553.988,E2 -1553.988} C_VEL
LIN {X 0,Y 587.353,Z 437.915,A -85,B 0,C 180,E1 -1554.628,E2 -1554.628} C_VEL
LIN {X 0,Y 587.286,Z 437.829,A -85,B 0,C 180,E1 -1557.68,E2 -1557.68} C_VEL
LIN {X 0,Y 587.313,Z 437.826,A -85,B 0,C 180,E1 -1560.505,E2 -1560.505} C_VEL
LIN {X 0,Y 587.308,Z 437.822,A -85,B 0,C 180,E1 -1563.398,E2 -1563.398} C_VEL
LIN {X 0,Y 587.27,Z 437.833,A -85,B 0,C 180,E1 -1565.901,E2 -1565.901} C_VEL
LIN {X 0,Y 587.308,Z 437.826,A -85,B 0,C 180,E1 -1568.481,E2 -1568.481} C_VEL
LIN {X 0,Y 587.284,Z 437.822,A -85,B 0,C 180,E1 -1571.161,E2 -1571.161} C_VEL
LIN {X 0,Y 587.302,Z 437.833,A -85,B 0,C 180,E1 -1574.11,E2 -1574.11} C_VEL
LIN {X 0,Y 587.271,Z 437.826,A -85,B 0,C 180,E1 -1576.989,E2 -1576.989} C_VEL
LIN {X 0,Y 587.292,Z 437.832,A -85,B 0,C 180,E1 -1579.984,E2 -1579.984} C_VEL
LIN {X 0,Y 587.304,Z 437.827,A -85,B 0,C 180,E1 -1582.389,E2 -1582.389} C_VEL
LIN {X 0,Y 587.32,Z 437.822,A -85,B 0,C 180,E1 -1585.655,E2 -1585.655} C_VEL
LIN {X 0,Y 587.33,Z 437.827,A -85,B 0,C 180,E1 -1588.23,E2 -1588.23} C_VEL
LIN {X 0,Y 587.294,Z 437.823,A -85,B 0,C 180,E1 -1590.875,E2 -1590.875} C_VEL
LIN {X 0,Y 587.298,Z 437.826,A -85,B 0,C 180,E1 -1593.83,E2 -1593.83} C_VEL
LIN {X 0,Y 587.296,Z 437.824,A -85,B 0,C 180,E1 -1596.739,E2 -1596.739} C_VEL
LIN {X 0,Y 587.298,Z 437.826,A -85,B 0,C 180,E1 -1599.693,E2 -1599.693} C_VEL
LIN {X 0,Y 587.267,Z 437.828,A -85,B 0,C 180,E1 -1602.591,E2 -1602.591} C_VEL
LIN {X 0,Y 587.308,Z 437.822,A -85,B 0,C 180,E1 -1605.445,E2 -1605.445} C_VEL
LIN {X 0,Y 587.31,Z 437.827,A -85,B 0,C 180,E1 -1608.262,E2 -1608.262} C_VEL
LIN {X 0,Y 587.27,Z 437.823,A -85,B 0,C 180,E1 -1611.049,E2 -1611.049} C_VEL
LIN {X 0,Y 587.303,Z 437.827,A -85,B 0,C 180,E1 -1613.816,E2 -1613.816} C_VEL
LIN {X 0,Y 587.296,Z 437.83,A -85,B 0,C 180,E1 -1615.882,E2 -1615.882} C_VEL
LIN {X 0,Y 587.366,Z 437.822,A -85,B 0,C 180,E1 -1617.942,E2 -1617.942} C_VEL
LIN {X 0,Y 587.374,Z 437.821,A -85,B 0,C 180,E1 -1619.999,E2 -1619.999} C_VEL
LIN {X 0,Y 587.327,Z 437.819,A -85,B 0,C 180,E1 -1622.742,E2 -1622.742} C_VEL
LIN {X 0,Y 587.316,Z 437.822,A -85,B 0,C 180,E1 -1625.492,E2 -1625.492} C_VEL
LIN {X 0,Y 587.32,Z 437.825,A -85,B 0,C 180,E1 -1628.255,E2 -1628.255} C_VEL
LIN {X 0,Y 587.288,Z 437.822,A -85,B 0,C 180,E1 -1631.106,E2 -1631.106} C_VEL
LIN {X 0,Y 587.336,Z 437.824,A -85,B 0,C 180,E1 -1633.845,E2 -1633.845} C_VEL
LIN {X 0,Y 587.275,Z 437.825,A -85,B 0,C 180,E1 -1636.792,E2 -1636.792} C_VEL
LIN {X 0,Y 587.263,Z 437.831,A -85,B 0,C 180,E1 -1638.274,E2 -1638.274} C_VEL
LIN {X 0,Y 586.597,Z 437.91,A -85,B 0,C 180,E1 -1638.846,E2 -1638.846} C_VEL
LIN {X 0,Y 583.749,Z 438.267,A -85,B 0,C 180,E1 -1639.775,E2 -1639.775} C_VEL
LIN {X 0,Y 581.353,Z 438.565,A -85,B 0,C 180,E1 -1640.522,E2 -1640.522} C_VEL
LIN {X 0,Y 580.339,Z 438.689,A -85,B 0,C 180,E1 -1641.099,E2 -1641.099} C_VEL
LIN {X 0,Y 580.263,Z 438.698,A -85,B 0,C 180,E1 -1641.294,E2 -1641.294} C_VEL
LIN {X 0,Y 580.246,Z 438.704,A -85,B 0,C 180,E1 -1643.558,E2 -1643.558} C_VEL
LIN {X 0,Y 580.241,Z 438.705,A -85,B 0,C 180,E1 -1646.325,E2 -1646.325} C_VEL
LIN {X 0,Y 580.239,Z 438.702,A -85,B 0,C 180,E1 -1649.3,E2 -1649.3} C_VEL
LIN {X 0,Y 580.264,Z 438.706,A -85,B 0,C 180,E1 -1652.201,E2 -1652.201} C_VEL
LIN {X 0,Y 580.257,Z 438.699,A -85,B 0,C 180,E1 -1654.697,E2 -1654.697} C_VEL
LIN {X 0,Y 580.252,Z 438.701,A -85,B 0,C 180,E1 -1657.27,E2 -1657.27} C_VEL
LIN {X 0,Y 580.266,Z 438.704,A -85,B 0,C 180,E1 -1660.268,E2 -1660.268} C_VEL
LIN {X 0,Y 580.234,Z 438.704,A -85,B 0,C 180,E1 -1662.708,E2 -1662.708} C_VEL
LIN {X 0,Y 580.235,Z 438.705,A -85,B 0,C 180,E1 -1665.61,E2 -1665.61} C_VEL
LIN {X 0,Y 580.224,Z 438.708,A -85,B 0,C 180,E1 -1668.227,E2 -1668.227} C_VEL
LIN {X 0,Y 580.245,Z 438.701,A -85,B 0,C 180,E1 -1670.963,E2 -1670.963} C_VEL
LIN {X 0,Y 580.216,Z 438.708,A -85,B 0,C 180,E1 -1673.593,E2 -1673.593} C_VEL
LIN {X 0,Y 580.251,Z 438.709,A -85,B 0,C 180,E1 -1676.141,E2 -1676.141} C_VEL
LIN {X 0,Y 580.247,Z 438.703,A -85,B 0,C 180,E1 -1678.613,E2 -1678.613} C_VEL
LIN {X 0,Y 580.23,Z 438.701,A -85,B 0,C 180,E1 -1681.021,E2 -1681.021} C_VEL
LIN {X 0,Y 580.244,Z 438.706,A -85,B 0,C 180,E1 -1683.672,E2 -1683.672} C_VEL
LIN {X 0,Y 580.24,Z 438.706,A -85,B 0,C 180,E1 -1686.441,E2 -1686.441} C_VEL
LIN {X 0,Y 580.236,Z 438.705,A -85,B 0,C 180,E1 -1689.436,E2 -1689.436} C_VEL
LIN {X 0,Y 580.223,Z 438.709,A -85,B 0,C 180,E1 -1691.644,E2 -1691.644} C_VEL
LIN {X 0,Y 580.25,Z 438.704,A -85,B 0,C 180,E1 -1694.546,E2 -1694.546} C_VEL
LIN {X 0,Y 580.22,Z 438.706,A -85,B 0,C 180,E1 -1696.695,E2 -1696.695} C_VEL
LIN {X 0,Y 580.249,Z 438.702,A -85,B 0,C 180,E1 -1698.826,E2 -1698.826} C_VEL
LIN {X 0,Y 580.284,Z 438.702,A -85,B 0,C 180,E1 -1701.643,E2 -1701.643} C_VEL
LIN {X 0,Y 580.28,Z 438.701,A -85,B 0,C 180,E1 -1704.44,E2 -1704.44} C_VEL
LIN {X 0,Y 580.286,Z 438.697,A -85,B 0,C 180,E1 -1707.223,E2 -1707.223} C_VEL
LIN {X 0,Y 580.334,Z 438.701,A -85,B 0,C 180,E1 -1710,E2 -1710} C_VEL
LIN {X 0,Y 580.286,Z 438.697,A -85,B 0,C 180,E1 -1712.777,E2 -1712.777} C_VEL
LIN {X 0,Y 580.28,Z 438.701,A -85,B 0,C 180,E1 -1715.56,E2 -1715.56} C_VEL
LIN {X 0,Y 580.284,Z 438.702,A -85,B 0,C 180,E1 -1718.357,E2 -1718.357} C_VEL
LIN {X 0,Y 580.249,Z 438.702,A -85,B 0,C 180,E1 -1721.174,E2 -1721.174} C_VEL
LIN {X 0,Y 580.291,Z 438.706,A -85,B 0,C 180,E1 -1724.018,E2 -1724.018} C_VEL
LIN {X 0,Y 580.232,Z 438.704,A -85,B 0,C 180,E1 -1726.9,E2 -1726.9} C_VEL
LIN {X 0,Y 580.255,Z 438.708,A -85,B 0,C 180,E1 -1729.824,E2 -1729.824} C_VEL
LIN {X 0,Y 580.258,Z 438.7,A -85,B 0,C 180,E1 -1732.804,E2 -1732.804} C_VEL
LIN {X 0,Y 580.228,Z 438.704,A -85,B 0,C 180,E1 -1735.083,E2 -1735.083} C_VEL
LIN {X 0,Y 580.231,Z 438.712,A -85,B 0,C 180,E1 -1737.85,E2 -1737.85} C_VEL
LIN {X 0,Y 580.25,Z 438.701,A -85,B 0,C 180,E1 -1740.692,E2 -1740.692} C_VEL
LIN {X 0,Y 580.252,Z 438.701,A -85,B 0,C 180,E1 -1743.312,E2 -1743.312} C_VEL
LIN {X 0,Y 580.206,Z 438.71,A -85,B 0,C 180,E1 -1745.754,E2 -1745.754} C_VEL
LIN {X 0,Y 580.261,Z 438.707,A -85,B 0,C 180,E1 -1748.148,E2 -1748.148} C_VEL
LIN {X 0,Y 580.224,Z 438.701,A -85,B 0,C 180,E1 -1750.849,E2 -1750.849} C_VEL
LIN {X 0,Y 580.218,Z 438.706,A -85,B 0,C 180,E1 -1753.663,E2 -1753.663} C_VEL
LIN {X 0,Y 580.219,Z 438.709,A -85,B 0,C 180,E1 -1756.339,E2 -1756.339} C_VEL
LIN {X 0,Y 580.258,Z 438.698,A -85,B 0,C 180,E1 -1759.155,E2 -1759.155} C_VEL
LIN {X 0,Y 580.264,Z 438.709,A -85,B 0,C 180,E1 -1761.93,E2 -1761.93} C_VEL
LIN {X 0,Y 580.206,Z 438.707,A -85,B 0,C 180,E1 -1764.451,E2 -1764.451} C_VEL
LIN {X 0,Y 580.229,Z 438.703,A -85,B 0,C 180,E1 -1766.973,E2 -1766.973} C_VEL
LIN {X 0,Y 580.265,Z 438.701,A -85,B 0,C 180,E1 -1769.425,E2 -1769.425} C_VEL
LIN {X 0,Y 580.236,Z 438.707,A -85,B 0,C 180,E1 -1772.152,E2 -1772.152} C_VEL
LIN {X 0,Y 580.233,Z 438.702,A -85,B 0,C 180,E1 -1774.918,E2 -1774.918} C_VEL
LIN {X 0,Y 580.264,Z 438.699,A -85,B 0,C 180,E1 -1777.198,E2 -1777.198} C_VEL
LIN {X 0,Y 580.243,Z 438.703,A -85,B 0,C 180,E1 -1779.437,E2 -1779.437} C_VEL
LIN {X 0,Y 580.229,Z 438.706,A -85,B 0,C 180,E1 -1782.375,E2 -1782.375} C_VEL
LIN {X 0,Y 580.256,Z 438.701,A -85,B 0,C 180,E1 -1785.266,E2 -1785.266} C_VEL
LIN {X 0,Y 580.279,Z 438.702,A -85,B 0,C 180,E1 -1788.119,E2 -1788.119} C_VEL
LIN {X 0,Y 580.227,Z 438.701,A -85,B 0,C 180,E1 -1790.942,E2 -1790.942} C_VEL
LIN {X 0,Y 580.257,Z 438.706,A -85,B 0,C 180,E1 -1793.743,E2 -1793.743} C_VEL
LIN {X 0,Y 580.252,Z 438.709,A -85,B 0,C 180,E1 -1795.834,E2 -1795.834} C_VEL
LIN {X 0,Y 580.332,Z 438.698,A -85,B 0,C 180,E1 -1797.919,E2 -1797.919} C_VEL
LIN {X 0,Y 580.342,Z 438.696,A -85,B 0,C 180,E1 -1800.001,E2 -1800.001} C_VEL
LIN {X 0,Y 580.293,Z 438.695,A -85,B 0,C 180,E1 -1802.778,E2 -1802.778} C_VEL
LIN {X 0,Y 580.29,Z 438.7,A -85,B 0,C 180,E1 -1805.561,E2 -1805.561} C_VEL
LIN {X 0,Y 580.288,Z 438.696,A -85,B 0,C 180,E1 -1808.358,E2 -1808.358} C_VEL
LIN {X 0,Y 580.263,Z 438.698,A -85,B 0,C 180,E1 -1811.175,E2 -1811.175} C_VEL
LIN {X 0,Y 580.296,Z 438.703,A -85,B 0,C 180,E1 -1814.019,E2 -1814.019} C_VEL
LIN {X 0,Y 580.224,Z 438.702,A -85,B 0,C 180,E1 -1816.901,E2 -1816.901} C_VEL
LIN {X 0,Y 580.244,Z 438.707,A -85,B 0,C 180,E1 -1819.825,E2 -1819.825} C_VEL
LIN {X 0,Y 580.241,Z 438.709,A -85,B 0,C 180,E1 -1822.055,E2 -1822.055} C_VEL
LIN {X 0,Y 580.251,Z 438.7,A -85,B 0,C 180,E1 -1824.716,E2 -1824.716} C_VEL
LIN {X 0,Y 580.235,Z 438.702,A -85,B 0,C 180,E1 -1827.405,E2 -1827.405} C_VEL
LIN {X 0,Y 580.255,Z 438.708,A -85,B 0,C 180,E1 -1829.775,E2 -1829.775} C_VEL
LIN {X 0,Y 580.274,Z 438.702,A -85,B 0,C 180,E1 -1832.203,E2 -1832.203} C_VEL
LIN {X 0,Y 580.265,Z 438.698,A -85,B 0,C 180,E1 -1834.699,E2 -1834.699} C_VEL
LIN {X 0,Y 580.261,Z 438.701,A -85,B 0,C 180,E1 -1837.272,E2 -1837.272} C_VEL
LIN {X 0,Y 580.247,Z 438.705,A -85,B 0,C 180,E1 -1840.266,E2 -1840.266} C_VEL
LIN {X 0,Y 580.242,Z 438.702,A -85,B 0,C 180,E1 -1842.71,E2 -1842.71} C_VEL
LIN {X 0,Y 580.247,Z 438.706,A -85,B 0,C 180,E1 -1845.612,E2 -1845.612} C_VEL
LIN {X 0,Y 580.236,Z 438.705,A -85,B 0,C 180,E1 -1848.228,E2 -1848.228} C_VEL
LIN {X 0,Y 580.258,Z 438.7,A -85,B 0,C 180,E1 -1850.964,E2 -1850.964} C_VEL
LIN {X 0,Y 580.22,Z 438.709,A -85,B 0,C 180,E1 -1853.593,E2 -1853.593} C_VEL
LIN {X 0,Y 580.262,Z 438.705,A -85,B 0,C 180,E1 -1856.142,E2 -1856.142} C_VEL
LIN {X 0,Y 580.239,Z 438.704,A -85,B 0,C 180,E1 -1858.613,E2 -1858.613} C_VEL
LIN {X 0,Y 580.243,Z 438.703,A -85,B 0,C 180,E1 -1861.021,E2 -1861.021} C_VEL
LIN {X 0,Y 580.245,Z 438.709,A -85,B 0,C 180,E1 -1863.676,E2 -1863.676} C_VEL
LIN {X 0,Y 580.302,Z 438.866,A -85,B 0,C 180,E1 -1865.246,E2 -1865.246} C_VEL
LIN {X 0,Y 580.807,Z 443.255,A -85,B 0,C 180,E1 -1866.086,E2 -1866.086} C_VEL
LIN {X 0,Y 580.606,Z 458.025,A -85,B 0,C 180,E1 -1868.758,E2 -1868.758} C_VEL
LIN {X 0,Y 580.514,Z 473.263,A -85,B 0,C 180,E1 -1871.471,E2 -1871.471} C_VEL
LIN {X 0,Y 580.384,Z 487.75,A -85,B 0,C 180,E1 -1874.009,E2 -1874.009} C_VEL
LIN {X 0,Y 580.345,Z 501.236,A -85,B 0,C 180,E1 -1876.319,E2 -1876.319} C_VEL
LIN {X 0,Y 580.681,Z 503.732,A -85,B 0,C 180,E1 -1876.394,E2 -1876.394} C_VEL
LIN {X 0,Y 580.936,Z 509.098,A -85,B 0,C 180,E1 -1876.467,E2 -1876.467} C_VEL
LIN {X 0,Y 580.786,Z 607.755,A -85,B 0,C 180,E1 -1877.708,E2 -1877.708} C_VEL
LIN {X 0,Y 580.729,Z 620.494,A -85,B 0,C 180,E1 -1877.995,E2 -1877.995} C_VEL
LIN {X 0,Y 580.636,Z 634.48,A -85,B 0,C 180,E1 -1878.48,E2 -1878.48} C_VEL
LIN {X 0,Y 580.563,Z 645.573,A -85,B 0,C 180,E1 -1879.009,E2 -1879.009} C_VEL
LIN {X 0,Y 580.458,Z 655.865,A -85,B 0,C 180,E1 -1879.624,E2 -1879.624} C_VEL
LIN {X 0,Y 580.374,Z 665.443,A -85,B 0,C 180,E1 -1880.327,E2 -1880.327} C_VEL
LIN {X 0,Y 580.305,Z 674.333,A -85,B 0,C 180,E1 -1881.117,E2 -1881.117} C_VEL
LIN {X 0,Y 580.222,Z 683.962,A -85,B 0,C 180,E1 -1882.168,E2 -1882.168} C_VEL
LIN {X 0,Y 580.151,Z 691.669,A -85,B 0,C 180,E1 -1883.226,E2 -1883.226} C_VEL
LIN {X 0,Y 580.161,Z 696.853,A -85,B 0,C 180,E1 -1884.09,E2 -1884.09} C_VEL
LIN {X 0,Y 580.053,Z 701.926,A -85,B 0,C 180,E1 -1885.135,E2 -1885.135} C_VEL
LIN {X 0,Y 580.11,Z 705.869,A -85,B 0,C 180,E1 -1886.179,E2 -1886.179} C_VEL
LIN {X 0,Y 580.043,Z 708.784,A -85,B 0,C 180,E1 -1887.222,E2 -1887.222} C_VEL
LIN {X 0,Y 580.04,Z 710.207,A -85,B 0,C 180,E1 -1887.917,E2 -1887.917} C_VEL
LIN {X 0,Y 580.04,Z 711.781,A -85,B 0,C 180,E1 -1889.306,E2 -1889.306} C_VEL
LIN {X 0,Y 580.037,Z 712,A -85,B 0,C 180,E1 -1890,E2 -1890} C_VEL
LIN {X 0,Y 580.046,Z 711.182,A -85,B 0,C 180,E1 -1891.389,E2 -1891.389} C_VEL
LIN {X 0,Y 580.04,Z 710.207,A -85,B 0,C 180,E1 -1892.083,E2 -1892.083} C_VEL
LIN {X 0,Y 580.043,Z 708.784,A -85,B 0,C 180,E1 -1892.778,E2 -1892.778} C_VEL
LIN {X 0,Y 580.11,Z 705.869,A -85,B 0,C 180,E1 -1893.821,E2 -1893.821} C_VEL
LIN {X 0,Y 580.053,Z 701.926,A -85,B 0,C 180,E1 -1894.865,E2 -1894.865} C_VEL
LIN {X 0,Y 580.161,Z 696.853,A -85,B 0,C 180,E1 -1895.91,E2 -1895.91} C_VEL
LIN {X 0,Y 580.185,Z 689.241,A -85,B 0,C 180,E1 -1897.132,E2 -1897.132} C_VEL
LIN {X 0,Y 580.251,Z 680.959,A -85,B 0,C 180,E1 -1898.182,E2 -1898.182} C_VEL
LIN {X 0,Y 580.308,Z 672.49,A -85,B 0,C 180,E1 -1899.058,E2 -1899.058} C_VEL
LIN {X 0,Y 580.392,Z 663.252,A -85,B 0,C 180,E1 -1899.848,E2 -1899.848} C_VEL
LIN {X 0,Y 580.536,Z 651.775,A -85,B 0,C 180,E1 -1900.639,E2 -1900.639} C_VEL
LIN {X 0,Y 580.594,Z 640.334,A -85,B 0,C 180,E1 -1901.258,E2 -1901.258} C_VEL
LIN {X 0,Y 580.681,Z 628.675,A -85,B 0,C 180,E1 -1901.74,E2 -1901.74} C_VEL
LIN {X 0,Y 580.767,Z 617.092,A -85,B 0,C 180,E1 -1902.093,E2 -1902.093} C_VEL
LIN {X 0,Y 580.79,Z 605.107,A -85,B 0,C 180,E1 -1902.336,E2 -1902.336} C_VEL
LIN {X 0,Y 580.817,Z 504.514,A -85,B 0,C 180,E1 -1903.593,E2 -1903.593} C_VEL
LIN {X 0,Y 580.388,Z 501.549,A -85,B 0,C 180,E1 -1903.658,E2 -1903.658} C_VEL
LIN {X 0,Y 580.336,Z 499.133,A -85,B 0,C 180,E1 -1904.017,E2 -1904.017} C_VEL
LIN {X 0,Y 580.42,Z 482.273,A -85,B 0,C 180,E1 -1906.947,E2 -1906.947} C_VEL
LIN {X 0,Y 580.561,Z 467.984,A -85,B 0,C 180,E1 -1909.464,E2 -1909.464} C_VEL
LIN {X 0,Y 580.719,Z 451.533,A -85,B 0,C 180,E1 -1912.409,E2 -1912.409} C_VEL
LIN {X 0,Y 580.701,Z 441.185,A -85,B 0,C 180,E1 -1914.298,E2 -1914.298} C_VEL
LIN {X 0,Y 580.272,Z 438.765,A -85,B 0,C 180,E1 -1914.809,E2 -1914.809} C_VEL
LIN {X 0,Y 580.233,Z 438.71,A -85,B 0,C 180,E1 -1917.846,E2 -1917.846} C_VEL
LIN {X 0,Y 580.257,Z 438.703,A -85,B 0,C 180,E1 -1920.689,E2 -1920.689} C_VEL
LIN {X 0,Y 580.269,Z 438.698,A -85,B 0,C 180,E1 -1923.31,E2 -1923.31} C_VEL
LIN {X 0,Y 580.218,Z 438.709,A -85,B 0,C 180,E1 -1925.752,E2 -1925.752} C_VEL
LIN {X 0,Y 580.275,Z 438.708,A -85,B 0,C 180,E1 -1928.147,E2 -1928.147} C_VEL
LIN {X 0,Y 580.235,Z 438.701,A -85,B 0,C 180,E1 -1930.848,E2 -1930.848} C_VEL
LIN {X 0,Y 580.232,Z 438.706,A -85,B 0,C 180,E1 -1933.662,E2 -1933.662} C_VEL
LIN {X 0,Y 580.221,Z 438.707,A -85,B 0,C 180,E1 -1936.615,E2 -1936.615} C_VEL
LIN {X 0,Y 580.235,Z 438.702,A -85,B 0,C 180,E1 -1939.15,E2 -1939.15} C_VEL
LIN {X 0,Y 580.267,Z 438.705,A -85,B 0,C 180,E1 -1941.929,E2 -1941.929} C_VEL
LIN {X 0,Y 580.215,Z 438.708,A -85,B 0,C 180,E1 -1944.449,E2 -1944.449} C_VEL
LIN {X 0,Y 580.238,Z 438.701,A -85,B 0,C 180,E1 -1946.971,E2 -1946.971} C_VEL
LIN {X 0,Y 580.273,Z 438.699,A -85,B 0,C 180,E1 -1949.423,E2 -1949.423} C_VEL
LIN {X 0,Y 580.235,Z 438.709,A -85,B 0,C 180,E1 -1952.152,E2 -1952.152} C_VEL
LIN {X 0,Y 580.241,Z 438.701,A -85,B 0,C 180,E1 -1954.916,E2 -1954.916} C_VEL
LIN {X 0,Y 580.271,Z 438.698,A -85,B 0,C 180,E1 -1957.196,E2 -1957.196} C_VEL
LIN {X 0,Y 580.241,Z 438.702,A -85,B 0,C 180,E1 -1959.435,E2 -1959.435} C_VEL
LIN {X 0,Y 580.234,Z 438.706,A -85,B 0,C 180,E1 -1962.373,E2 -1962.373} C_VEL
LIN {X 0,Y 580.256,Z 438.7,A -85,B 0,C 180,E1 -1965.264,E2 -1965.264} C_VEL
LIN {X 0,Y 580.282,Z 438.705,A -85,B 0,C 180,E1 -1968.117,E2 -1968.117} C_VEL
LIN {X 0,Y 580.229,Z 438.7,A -85,B 0,C 180,E1 -1970.939,E2 -1970.939} C_VEL
LIN {X 0,Y 580.255,Z 438.704,A -85,B 0,C 180,E1 -1973.741,E2 -1973.741} C_VEL
LIN {X 0,Y 580.249,Z 438.707,A -85,B 0,C 180,E1 -1975.832,E2 -1975.832} C_VEL
LIN {X 0,Y 580.335,Z 438.697,A -85,B 0,C 180,E1 -1977.917,E2 -1977.917} C_VEL
LIN {X 0,Y 580.342,Z 438.696,A -85,B 0,C 180,E1 -1979.999,E2 -1979.999} C_VEL
LIN {X 0,Y 580.295,Z 438.695,A -85,B 0,C 180,E1 -1982.776,E2 -1982.776} C_VEL
LIN {X 0,Y 580.286,Z 438.699,A -85,B 0,C 180,E1 -1985.559,E2 -1985.559} C_VEL
LIN {X 0,Y 580.286,Z 438.699,A -85,B 0,C 180,E1 -1988.355,E2 -1988.355} C_VEL
LIN {X 0,Y 580.259,Z 438.697,A -85,B 0,C 180,E1 -1991.173,E2 -1991.173} C_VEL
LIN {X 0,Y 580.299,Z 438.704,A -85,B 0,C 180,E1 -1994.016,E2 -1994.016} C_VEL
LIN {X 0,Y 580.222,Z 438.703,A -85,B 0,C 180,E1 -1996.899,E2 -1996.899} C_VEL
LIN {X 0,Y 580.256,Z 438.703,A -85,B 0,C 180,E1 -1999.823,E2 -1999.823} C_VEL
LIN {X 0,Y 580.263,Z 438.698,A -85,B 0,C 180,E1 -2001.294,E2 -2001.294} C_VEL
LIN {X 0,Y 579.609,Z 438.788,A -85,B 0,C 180,E1 -2001.873,E2 -2001.873} C_VEL
LIN {X 0,Y 576.732,Z 439.144,A -85,B 0,C 180,E1 -2002.813,E2 -2002.813} C_VEL
LIN {X 0,Y 574.299,Z 439.447,A -85,B 0,C 180,E1 -2003.569,E2 -2003.569} C_VEL
LIN {X 0,Y 573.267,Z 439.579,A -85,B 0,C 180,E1 -2004.153,E2 -2004.153} C_VEL
LIN {X 0,Y 573.19,Z 439.582,A -85,B 0,C 180,E1 -2004.351,E2 -2004.351} C_VEL
LIN {X 0,Y 573.169,Z 439.58,A -85,B 0,C 180,E1 -2006.978,E2 -2006.978} C_VEL
LIN {X 0,Y 573.192,Z 439.581,A -85,B 0,C 180,E1 -2009.479,E2 -2009.479} C_VEL
LIN {X 0,Y 573.217,Z 439.583,A -85,B 0,C 180,E1 -2012.224,E2 -2012.224} C_VEL
LIN {X 0,Y 573.202,Z 439.577,A -85,B 0,C 180,E1 -2014.767,E2 -2014.767} C_VEL
LIN {X 0,Y 573.203,Z 439.585,A -85,B 0,C 180,E1 -2017.808,E2 -2017.808} C_VEL
LIN {X 0,Y 573.231,Z 439.576,A -85,B 0,C 180,E1 -2020.524,E2 -2020.524} C_VEL
LIN {X 0,Y 573.181,Z 439.582,A -85,B 0,C 180,E1 -2023.362,E2 -2023.362} C_VEL
LIN {X 0,Y 573.187,Z 439.581,A -85,B 0,C 180,E1 -2026.335,E2 -2026.335} C_VEL
LIN {X 0,Y 573.176,Z 439.581,A -85,B 0,C 180,E1 -2028.539,E2 -2028.539} C_VEL
LIN {X 0,Y 573.214,Z 439.578,A -85,B 0,C 180,E1 -2031.297,E2 -2031.297} C_VEL
LIN {X 0,Y 573.166,Z 439.591,A -85,B 0,C 180,E1 -2034.022,E2 -2034.022} C_VEL
LIN {X 0,Y 573.204,Z 439.581,A -85,B 0,C 180,E1 -2036.514,E2 -2036.514} C_VEL
LIN {X 0,Y 573.201,Z 439.579,A -85,B 0,C 180,E1 -2039.119,E2 -2039.119} C_VEL
LIN {X 0,Y 573.185,Z 439.589,A -85,B 0,C 180,E1 -2041.98,E2 -2041.98} C_VEL
LIN {X 0,Y 573.192,Z 439.582,A -85,B 0,C 180,E1 -2044.587,E2 -2044.587} C_VEL
LIN {X 0,Y 573.2,Z 439.58,A -85,B 0,C 180,E1 -2046.899,E2 -2046.899} C_VEL
LIN {X 0,Y 573.21,Z 439.578,A -85,B 0,C 180,E1 -2049.172,E2 -2049.172} C_VEL
LIN {X 0,Y 573.179,Z 439.584,A -85,B 0,C 180,E1 -2051.41,E2 -2051.41} C_VEL
LIN {X 0,Y 573.189,Z 439.586,A -85,B 0,C 180,E1 -2054.351,E2 -2054.351} C_VEL
LIN {X 0,Y 573.184,Z 439.584,A -85,B 0,C 180,E1 -2056.528,E2 -2056.528} C_VEL
LIN {X 0,Y 573.228,Z 439.578,A -85,B 0,C 180,E1 -2059.403,E2 -2059.403} C_VEL
LIN {X 0,Y 573.202,Z 439.586,A -85,B 0,C 180,E1 -2062.249,E2 -2062.249} C_VEL
LIN {X 0,Y 573.258,Z 439.573,A -85,B 0,C 180,E1 -2065.077,E2 -2065.077} C_VEL
LIN {X 0,Y 573.296,Z 439.576,A -85,B 0,C 180,E1 -2067.892,E2 -2067.892} C_VEL
LIN {X 0,Y 573.302,Z 439.577,A -85,B 0,C 180,E1 -2070,E2 -2070} C_VEL
LIN {X 0,Y 573.254,Z 439.573,A -85,B 0,C 180,E1 -2072.811,E2 -2072.811} C_VEL
LIN {X 0,Y 573.25,Z 439.578,A -85,B 0,C 180,E1 -2075.629,E2 -2075.629} C_VEL
LIN {X 0,Y 573.226,Z 439.58,A -85,B 0,C 180,E1 -2078.46,E2 -2078.46} C_VEL
LIN {X 0,Y 573.218,Z 439.579,A -85,B 0,C 180,E1 -2081.313,E2 -2081.313} C_VEL
LIN {X 0,Y 573.253,Z 439.577,A -85,B 0,C 180,E1 -2084.42,E2 -2084.42} C_VEL
LIN {X 0,Y 573.175,Z 439.583,A -85,B 0,C 180,E1 -2087.114,E2 -2087.114} C_VEL
LIN {X 0,Y 573.248,Z 439.575,A -85,B 0,C 180,E1 -2089.33,E2 -2089.33} C_VEL
LIN {X 0,Y 573.198,Z 439.584,A -85,B 0,C 180,E1 -2092.339,E2 -2092.339} C_VEL
LIN {X 0,Y 573.186,Z 439.581,A -85,B 0,C 180,E1 -2094.865,E2 -2094.865} C_VEL
LIN {X 0,Y 573.167,Z 439.583,A -85,B 0,C 180,E1 -2096.98,E2 -2096.98} C_VEL
LIN {X 0,Y 573.188,Z 439.581,A -85,B 0,C 180,E1 -2099.481,E2 -2099.481} C_VEL
LIN {X 0,Y 573.213,Z 439.583,A -85,B 0,C 180,E1 -2102.225,E2 -2102.225} C_VEL
LIN {X 0,Y 573.2,Z 439.576,A -85,B 0,C 180,E1 -2104.769,E2 -2104.769} C_VEL
LIN {X 0,Y 573.201,Z 439.586,A -85,B 0,C 180,E1 -2107.81,E2 -2107.81} C_VEL
LIN {X 0,Y 573.184,Z 439.579,A -85,B 0,C 180,E1 -2110.53,E2 -2110.53} C_VEL
LIN {X 0,Y 573.18,Z 439.579,A -85,B 0,C 180,E1 -2113.364,E2 -2113.364} C_VEL
LIN {X 0,Y 573.188,Z 439.585,A -85,B 0,C 180,E1 -2116.336,E2 -2116.336} C_VEL
LIN {X 0,Y 573.185,Z 439.581,A -85,B 0,C 180,E1 -2118.541,E2 -2118.541} C_VEL
LIN {X 0,Y 573.215,Z 439.578,A -85,B 0,C 180,E1 -2121.298,E2 -2121.298} C_VEL
LIN {X 0,Y 573.168,Z 439.59,A -85,B 0,C 180,E1 -2124.024,E2 -2124.024} C_VEL
LIN {X 0,Y 573.208,Z 439.579,A -85,B 0,C 180,E1 -2126.516,E2 -2126.516} C_VEL
LIN {X 0,Y 573.205,Z 439.579,A -85,B 0,C 180,E1 -2129.121,E2 -2129.121} C_VEL
LIN {X 0,Y 573.19,Z 439.587,A -85,B 0,C 180,E1 -2131.982,E2 -2131.982} C_VEL
LIN {X 0,Y 573.195,Z 439.58,A -85,B 0,C 180,E1 -2134.589,E2 -2134.589} C_VEL
LIN {X 0,Y 573.207,Z 439.578,A -85,B 0,C 180,E1 -2136.901,E2 -2136.901} C_VEL
LIN {X 0,Y 573.217,Z 439.576,A -85,B 0,C 180,E1 -2139.174,E2 -2139.174} C_VEL
LIN {X 0,Y 573.19,Z 439.586,A -85,B 0,C 180,E1 -2142.151,E2 -2142.151} C_VEL
LIN {X 0,Y 573.204,Z 439.578,A -85,B 0,C 180,E1 -2145.081,E2 -2145.081} C_VEL
LIN {X 0,Y 573.225,Z 439.583,A -85,B 0,C 180,E1 -2147.971,E2 -2147.971} C_VEL
LIN {X 0,Y 573.193,Z 439.577,A -85,B 0,C 180,E1 -2150.829,E2 -2150.829} C_VEL
LIN {X 0,Y 573.215,Z 439.582,A -85,B 0,C 180,E1 -2153.666,E2 -2153.666} C_VEL
LIN {X 0,Y 573.207,Z 439.586,A -85,B 0,C 180,E1 -2155.782,E2 -2155.782} C_VEL
LIN {X 0,Y 573.301,Z 439.574,A -85,B 0,C 180,E1 -2157.893,E2 -2157.893} C_VEL
LIN {X 0,Y 573.311,Z 439.571,A -85,B 0,C 180,E1 -2160.001,E2 -2160.001} C_VEL
LIN {X 0,Y 573.262,Z 439.571,A -85,B 0,C 180,E1 -2162.812,E2 -2162.812} C_VEL
LIN {X 0,Y 573.259,Z 439.577,A -85,B 0,C 180,E1 -2165.629,E2 -2165.629} C_VEL
LIN {X 0,Y 573.229,Z 439.573,A -85,B 0,C 180,E1 -2168.461,E2 -2168.461} C_VEL
LIN {X 0,Y 573.231,Z 439.574,A -85,B 0,C 180,E1 -2171.314,E2 -2171.314} C_VEL
LIN {X 0,Y 573.238,Z 439.576,A -85,B 0,C 180,E1 -2174.409,E2 -2174.409} C_VEL
LIN {X 0,Y 573.173,Z 439.58,A -85,B 0,C 180,E1 -2177.115,E2 -2177.115} C_VEL
LIN {X 0,Y 573.188,Z 439.587,A -85,B 0,C 180,E1 -2180.08,E2 -2180.08} C_VEL
LIN {X 0,Y 573.21,Z 439.581,A -85,B 0,C 180,E1 -2182.34,E2 -2182.34} C_VEL
LIN {X 0,Y 573.204,Z 439.58,A -85,B 0,C 180,E1 -2185.413,E2 -2185.413} C_VEL
LIN {X 0,Y 573.189,Z 439.588,A -85,B 0,C 180,E1 -2188.018,E2 -2188.018} C_VEL
LIN {X 0,Y 573.215,Z 439.577,A -85,B 0,C 180,E1 -2190.881,E2 -2190.881} C_VEL
LIN {X 0,Y 573.24,Z 439.576,A -85,B 0,C 180,E1 -2193.521,E2 -2193.521} C_VEL
LIN {X 0,Y 573.18,Z 439.589,A -85,B 0,C 180,E1 -2196.055,E2 -2196.055} C_VEL
LIN {X 0,Y 573.212,Z 439.577,A -85,B 0,C 180,E1 -2198.705,E2 -2198.705} C_VEL
LIN {X 0,Y 573.185,Z 439.586,A -85,B 0,C 180,E1 -2201.588,E2 -2201.588} C_VEL
LIN {X 0,Y 573.204,Z 439.581,A -85,B 0,C 180,E1 -2204.337,E2 -2204.337} C_VEL
LIN {X 0,Y 573.193,Z 439.58,A -85,B 0,C 180,E1 -2206.637,E2 -2206.637} C_VEL
LIN {X 0,Y 573.2,Z 439.58,A -85,B 0,C 180,E1 -2209.481,E2 -2209.481} C_VEL
LIN {X 0,Y 573.213,Z 439.582,A -85,B 0,C 180,E1 -2212.191,E2 -2212.191} C_VEL
LIN {X 0,Y 573.212,Z 439.579,A -85,B 0,C 180,E1 -2215.233,E2 -2215.233} C_VEL
LIN {X 0,Y 573.215,Z 439.583,A -85,B 0,C 180,E1 -2218.183,E2 -2218.183} C_VEL
LIN {X 0,Y 573.219,Z 439.579,A -85,B 0,C 180,E1 -2220.632,E2 -2220.632} C_VEL
LIN {X 0,Y 573.188,Z 439.587,A -85,B 0,C 180,E1 -2223.518,E2 -2223.518} C_VEL
LIN {X 0,Y 573.232,Z 439.754,A -85,B 0,C 180,E1 -2225.094,E2 -2225.094} C_VEL
LIN {X 0,Y 573.862,Z 444.285,A -85,B 0,C 180,E1 -2225.971,E2 -2225.971} C_VEL
LIN {X 0,Y 573.645,Z 460.277,A -85,B 0,C 180,E1 -2228.898,E2 -2228.898} C_VEL
LIN {X 0,Y 573.501,Z 476.368,A -85,B 0,C 180,E1 -2231.791,E2 -2231.791} C_VEL
LIN {X 0,Y 573.306,Z 492.924,A -85,B 0,C 180,E1 -2234.719,E2 -2234.719} C_VEL
LIN {X 0,Y 573.32,Z 501.242,A -85,B 0,C 180,E1 -2236.148,E2 -2236.148} C_VEL
LIN {X 0,Y 573.632,Z 503.524,A -85,B 0,C 180,E1 -2236.221,E2 -2236.221} C_VEL
LIN {X 0,Y 574.081,Z 507.309,A -85,B 0,C 180,E1 -2236.279,E2 -2236.279} C_VEL
LIN {X 0,Y 573.863,Z 607.705,A -85,B 0,C 180,E1 -2237.557,E2 -2237.557} C_VEL
LIN {X 0,Y 573.81,Z 620.49,A -85,B 0,C 180,E1 -2237.848,E2 -2237.848} C_VEL
LIN {X 0,Y 573.685,Z 634.47,A -85,B 0,C 180,E1 -2238.339,E2 -2238.339} C_VEL
LIN {X 0,Y 573.588,Z 645.647,A -85,B 0,C 180,E1 -2238.878,E2 -2238.878} C_VEL
LIN {X 0,Y 573.469,Z 655.851,A -85,B 0,C 180,E1 -2239.497,E2 -2239.497} C_VEL
LIN {X 0,Y 573.36,Z 665.431,A -85,B 0,C 180,E1 -2240.208,E2 -2240.208} C_VEL
LIN {X 0,Y 573.254,Z 674.323,A -85,B 0,C 180,E1 -2241.007,E2 -2241.007} C_VEL
LIN {X 0,Y 573.161,Z 683.962,A -85,B 0,C 180,E1 -2242.071,E2 -2242.071} C_VEL
LIN {X 0,Y 573.071,Z 691.596,A -85,B 0,C 180,E1 -2243.13,E2 -2243.13} C_VEL
LIN {X 0,Y 573.073,Z 696.85,A -85,B 0,C 180,E1 -2244.017,E2 -2244.017} C_VEL
LIN {X 0,Y 572.962,Z 701.921,A -85,B 0,C 180,E1 -2245.074,E2 -2245.074} C_VEL
LIN {X 0,Y 573.015,Z 705.862,A -85,B 0,C 180,E1 -2246.132,E2 -2246.132} C_VEL
LIN {X 0,Y 572.959,Z 708.777,A -85,B 0,C 180,E1 -2247.188,E2 -2247.188} C_VEL
LIN {X 0,Y 572.939,Z 710.208,A -85,B 0,C 180,E1 -2247.891,E2 -2247.891} C_VEL
LIN {X 0,Y 572.941,Z 711.774,A -85,B 0,C 180,E1 -2249.297,E2 -2249.297} C_VEL
LIN {X 0,Y 572.938,Z 712,A -85,B 0,C 180,E1 -2250,E2 -2250} C_VEL
LIN {X 0,Y 572.946,Z 711.181,A -85,B 0,C 180,E1 -2251.406,E2 -2251.406} C_VEL
LIN {X 0,Y 572.939,Z 710.208,A -85,B 0,C 180,E1 -2252.109,E2 -2252.109} C_VEL
LIN {X 0,Y 572.959,Z 708.777,A -85,B 0,C 180,E1 -2252.812,E2 -2252.812} C_VEL
LIN {X 0,Y 573.015,Z 705.862,A -85,B 0,C 180,E1 -2253.868,E2 -2253.868} C_VEL
LIN {X 0,Y 572.962,Z 701.921,A -85,B 0,C 180,E1 -2254.926,E2 -2254.926} C_VEL
LIN {X 0,Y 573.073,Z 696.85,A -85,B 0,C 180,E1 -2255.983,E2 -2255.983} C_VEL
LIN {X 0,Y 573.114,Z 689.242,A -85,B 0,C 180,E1 -2257.221,E2 -2257.221} C_VEL
LIN {X 0,Y 573.199,Z 680.949,A -85,B 0,C 180,E1 -2258.283,E2 -2258.283} C_VEL
LIN {X 0,Y 573.287,Z 672.479,A -85,B 0,C 180,E1 -2259.17,E2 -2259.17} C_VEL
LIN {X 0,Y 573.398,Z 663.24,A -85,B 0,C 180,E1 -2259.97,E2 -2259.97} C_VEL
LIN {X 0,Y 573.552,Z 651.818,A -85,B 0,C 180,E1 -2260.767,E2 -2260.767} C_VEL
LIN {X 0,Y 573.603,Z 639.766,A -85,B 0,C 180,E1 -2261.422,E2 -2261.422} C_VEL
LIN {X 0,Y 573.714,Z 628.653,A -85,B 0,C 180,E1 -2261.885,E2 -2261.885} C_VEL
LIN {X 0,Y 573.84,Z 617.06,A -85,B 0,C 180,E1 -2262.241,E2 -2262.241} C_VEL
LIN {X 0,Y 573.868,Z 605.063,A -85,B 0,C 180,E1 -2262.488,E2 -2262.488} C_VEL
LIN {X 0,Y 573.948,Z 505.42,A -85,B 0,C 180,E1 -2263.748,E2 -2263.748} C_VEL
LIN {X 0,Y 573.34,Z 501.557,A -85,B 0,C 180,E1 -2263.829,E2 -2263.829} C_VEL
LIN {X 0,Y 573.296,Z 499.133,A -85,B 0,C 180,E1 -2264.192,E2 -2264.192} C_VEL
LIN {X 0,Y 573.409,Z 482.577,A -85,B 0,C 180,E1 -2267.107,E2 -2267.107} C_VEL
LIN {X 0,Y 573.578,Z 468.092,A -85,B 0,C 180,E1 -2269.691,E2 -2269.691} C_VEL
LIN {X 0,Y 573.748,Z 452.568,A -85,B 0,C 180,E1 -2272.506,E2 -2272.506} C_VEL
LIN {X 0,Y 573.825,Z 443.235,A -85,B 0,C 180,E1 -2274.223,E2 -2274.223} C_VEL
LIN {X 0,Y 573.228,Z 439.649,A -85,B 0,C 180,E1 -2274.948,E2 -2274.948} C_VEL
LIN {X 0,Y 573.213,Z 439.584,A -85,B 0,C 180,E1 -2277.769,E2 -2277.769} C_VEL
LIN {X 0,Y 573.222,Z 439.585,A -85,B 0,C 180,E1 -2280.177,E2 -2280.177} C_VEL
LIN {X 0,Y 573.223,Z 439.578,A -85,B 0,C 180,E1 -2282.647,E2 -2282.647} C_VEL
LIN {X 0,Y 573.18,Z 439.581,A -85,B 0,C 180,E1 -2285.189,E2 -2285.189} C_VEL
LIN {X 0,Y 573.213,Z 439.582,A -85,B 0,C 180,E1 -2287.809,E2 -2287.809} C_VEL
LIN {X 0,Y 573.2,Z 439.579,A -85,B 0,C 180,E1 -2290.528,E2 -2290.528} C_VEL
LIN {X 0,Y 573.193,Z 439.58,A -85,B 0,C 180,E1 -2293.363,E2 -2293.363} C_VEL
LIN {X 0,Y 573.194,Z 439.586,A -85,B 0,C 180,E1 -2296.336,E2 -2296.336} C_VEL
LIN {X 0,Y 573.186,Z 439.584,A -85,B 0,C 180,E1 -2298.538,E2 -2298.538} C_VEL
LIN {X 0,Y 573.212,Z 439.577,A -85,B 0,C 180,E1 -2301.295,E2 -2301.295} C_VEL
LIN {X 0,Y 573.179,Z 439.591,A -85,B 0,C 180,E1 -2304.022,E2 -2304.022} C_VEL
LIN {X 0,Y 573.22,Z 439.578,A -85,B 0,C 180,E1 -2306.514,E2 -2306.514} C_VEL
LIN {X 0,Y 573.215,Z 439.577,A -85,B 0,C 180,E1 -2309.119,E2 -2309.119} C_VEL
LIN {X 0,Y 573.189,Z 439.588,A -85,B 0,C 180,E1 -2311.982,E2 -2311.982} C_VEL
LIN {X 0,Y 573.204,Z 439.58,A -85,B 0,C 180,E1 -2314.587,E2 -2314.587} C_VEL
LIN {X 0,Y 573.21,Z 439.581,A -85,B 0,C 180,E1 -2317.66,E2 -2317.66} C_VEL
LIN {X 0,Y 573.188,Z 439.587,A -85,B 0,C 180,E1 -2319.92,E2 -2319.92} C_VEL
LIN {X 0,Y 573.188,Z 439.578,A -85,B 0,C 180,E1 -2323.012,E2 -2323.012} C_VEL
LIN {X 0,Y 573.242,Z 439.579,A -85,B 0,C 180,E1 -2325.805,E2 -2325.805} C_VEL
LIN {X 0,Y 573.222,Z 439.575,A -85,B 0,C 180,E1 -2328.763,E2 -2328.763} C_VEL
LIN {X 0,Y 573.229,Z 439.573,A -85,B 0,C 180,E1 -2331.539,E2 -2331.539} C_VEL
LIN {X 0,Y 573.259,Z 439.577,A -85,B 0,C 180,E1 -2334.371,E2 -2334.371} C_VEL
LIN {X 0,Y 573.304,Z 439.573,A -85,B 0,C 180,E1 -2337.891,E2 -2337.891} C_VEL
LIN {X 0,Y 573.311,Z 439.571,A -85,B 0,C 180,E1 -2339.999,E2 -2339.999} C_VEL
LIN {X 0,Y 573.263,Z 439.571,A -85,B 0,C 180,E1 -2342.81,E2 -2342.81} C_VEL
LIN {X 0,Y 573.255,Z 439.575,A -85,B 0,C 180,E1 -2345.627,E2 -2345.627} C_VEL
LIN {X 0,Y 573.227,Z 439.576,A -85,B 0,C 180,E1 -2348.459,E2 -2348.459} C_VEL
LIN {X 0,Y 573.227,Z 439.573,A -85,B 0,C 180,E1 -2351.312,E2 -2351.312} C_VEL
LIN {X 0,Y 573.24,Z 439.578,A -85,B 0,C 180,E1 -2354.41,E2 -2354.41} C_VEL
LIN {X 0,Y 573.17,Z 439.581,A -85,B 0,C 180,E1 -2357.113,E2 -2357.113} C_VEL
LIN {X 0,Y 573.213,Z 439.584,A -85,B 0,C 180,E1 -2360.077,E2 -2360.077} C_VEL
LIN {X 0,Y 573.204,Z 439.584,A -85,B 0,C 180,E1 -2362.338,E2 -2362.338} C_VEL
LIN {X 0,Y 573.19,Z 439.582,A -85,B 0,C 180,E1 -2364.351,E2 -2364.351} C_VEL
LIN {X 0,Y 572.547,Z 439.663,A -85,B 0,C 180,E1 -2364.937,E2 -2364.937} C_VEL
LIN {X 0,Y 569.709,Z 440.021,A -85,B 0,C 180,E1 -2365.889,E2 -2365.889} C_VEL
LIN {X 0,Y 567.287,Z 440.316,A -85,B 0,C 180,E1 -2366.654,E2 -2366.654} C_VEL
LIN {X 0,Y 566.232,Z 440.444,A -85,B 0,C 180,E1 -2367.245,E2 -2367.245} C_VEL
LIN {X 0,Y 566.139,Z 440.456,A -85,B 0,C 180,E1 -2367.445,E2 -2367.445} C_VEL
LIN {X 0,Y 566.153,Z 440.459,A -85,B 0,C 180,E1 -2370.593,E2 -2370.593} C_VEL
LIN {X 0,Y 566.149,Z 440.456,A -85,B 0,C 180,E1 -2373.105,E2 -2373.105} C_VEL
LIN {X 0,Y 566.123,Z 440.463,A -85,B 0,C 180,E1 -2375.693,E2 -2375.693} C_VEL
LIN {X 0,Y 566.186,Z 440.455,A -85,B 0,C 180,E1 -2378.556,E2 -2378.556} C_VEL
LIN {X 0,Y 566.139,Z 440.456,A -85,B 0,C 180,E1 -2381.141,E2 -2381.141} C_VEL
LIN {X 0,Y 566.142,Z 440.468,A -85,B 0,C 180,E1 -2384.039,E2 -2384.039} C_VEL
LIN {X 0,Y 566.136,Z 440.454,A -85,B 0,C 180,E1 -2387.088,E2 -2387.088} C_VEL
LIN {X 0,Y 566.171,Z 440.46,A -85,B 0,C 180,E1 -2390.317,E2 -2390.317} C_VEL
LIN {X 0,Y 566.168,Z 440.457,A -85,B 0,C 180,E1 -2392.6,E2 -2392.6} C_VEL
LIN {X 0,Y 566.163,Z 440.452,A -85,B 0,C 180,E1 -2395.179,E2 -2395.179} C_VEL
LIN {X 0,Y 566.192,Z 440.457,A -85,B 0,C 180,E1 -2397.741,E2 -2397.741} C_VEL
LIN {X 0,Y 566.141,Z 440.461,A -85,B 0,C 180,E1 -2400.336,E2 -2400.336} C_VEL
LIN {X 0,Y 566.161,Z 440.458,A -85,B 0,C 180,E1 -2403.456,E2 -2403.456} C_VEL
LIN {X 0,Y 566.146,Z 440.465,A -85,B 0,C 180,E1 -2405.817,E2 -2405.817} C_VEL
LIN {X 0,Y 566.173,Z 440.455,A -85,B 0,C 180,E1 -2408.901,E2 -2408.901} C_VEL
LIN {X 0,Y 566.167,Z 440.456,A -85,B 0,C 180,E1 -2411.171,E2 -2411.171} C_VEL
LIN {X 0,Y 566.154,Z 440.465,A -85,B 0,C 180,E1 -2414.151,E2 -2414.151} C_VEL
LIN {X 0,Y 566.153,Z 440.462,A -85,B 0,C 180,E1 -2416.358,E2 -2416.358} C_VEL
LIN {X 0,Y 566.197,Z 440.453,A -85,B 0,C 180,E1 -2419.27,E2 -2419.27} C_VEL
LIN {X 0,Y 566.171,Z 440.464,A -85,B 0,C 180,E1 -2422.152,E2 -2422.152} C_VEL
LIN {X 0,Y 566.233,Z 440.448,A -85,B 0,C 180,E1 -2425.016,E2 -2425.016} C_VEL
LIN {X 0,Y 566.265,Z 440.452,A -85,B 0,C 180,E1 -2427.866,E2 -2427.866} C_VEL
LIN {X 0,Y 566.27,Z 440.452,A -85,B 0,C 180,E1 -2430,E2 -2430} C_VEL
LIN {X 0,Y 566.222,Z 440.45,A -85,B 0,C 180,E1 -2432.846,E2 -2432.846} C_VEL
LIN {X 0,Y 566.22,Z 440.455,A -85,B 0,C 180,E1 -2435.699,E2 -2435.699} C_VEL
LIN {X 0,Y 566.177,Z 440.457,A -85,B 0,C 180,E1 -2438.566,E2 -2438.566} C_VEL
LIN {X 0,Y 566.175,Z 440.457,A -85,B 0,C 180,E1 -2441.456,E2 -2441.456} C_VEL
LIN {X 0,Y 566.207,Z 440.454,A -85,B 0,C 180,E1 -2444.502,E2 -2444.502} C_VEL
LIN {X 0,Y 566.141,Z 440.46,A -85,B 0,C 180,E1 -2447.333,E2 -2447.333} C_VEL
LIN {X 0,Y 566.18,Z 440.458,A -85,B 0,C 180,E1 -2449.582,E2 -2449.582} C_VEL
LIN {X 0,Y 566.164,Z 440.464,A -85,B 0,C 180,E1 -2451.864,E2 -2451.864} C_VEL
LIN {X 0,Y 566.146,Z 440.465,A -85,B 0,C 180,E1 -2454.183,E2 -2454.183} C_VEL
LIN {X 0,Y 566.154,Z 440.458,A -85,B 0,C 180,E1 -2456.652,E2 -2456.652} C_VEL
LIN {X 0,Y 566.142,Z 440.462,A -85,B 0,C 180,E1 -2459.772,E2 -2459.772} C_VEL
LIN {X 0,Y 566.161,Z 440.458,A -85,B 0,C 180,E1 -2462.426,E2 -2462.426} C_VEL
LIN {X 0,Y 566.145,Z 440.454,A -85,B 0,C 180,E1 -2464.987,E2 -2464.987} C_VEL
LIN {X 0,Y 566.168,Z 440.457,A -85,B 0,C 180,E1 -2467.463,E2 -2467.463} C_VEL
LIN {X 0,Y 566.144,Z 440.46,A -85,B 0,C 180,E1 -2470.204,E2 -2470.204} C_VEL
LIN {X 0,Y 566.131,Z 440.454,A -85,B 0,C 180,E1 -2473.06,E2 -2473.06} C_VEL
LIN {X 0,Y 566.14,Z 440.467,A -85,B 0,C 180,E1 -2476.054,E2 -2476.054} C_VEL
LIN {X 0,Y 566.139,Z 440.456,A -85,B 0,C 180,E1 -2478.859,E2 -2478.859} C_VEL
LIN {X 0,Y 566.186,Z 440.455,A -85,B 0,C 180,E1 -2481.444,E2 -2481.444} C_VEL
LIN {X 0,Y 566.123,Z 440.463,A -85,B 0,C 180,E1 -2484.307,E2 -2484.307} C_VEL
LIN {X 0,Y 566.149,Z 440.456,A -85,B 0,C 180,E1 -2486.895,E2 -2486.895} C_VEL
LIN {X 0,Y 566.153,Z 440.459,A -85,B 0,C 180,E1 -2489.407,E2 -2489.407} C_VEL
LIN {X 0,Y 566.136,Z 440.466,A -85,B 0,C 180,E1 -2491.855,E2 -2491.855} C_VEL
LIN {X 0,Y 566.164,Z 440.46,A -85,B 0,C 180,E1 -2494.25,E2 -2494.25} C_VEL
LIN {X 0,Y 566.154,Z 440.457,A -85,B 0,C 180,E1 -2496.721,E2 -2496.721} C_VEL
LIN {X 0,Y 566.18,Z 440.452,A -85,B 0,C 180,E1 -2498.903,E2 -2498.903} C_VEL
LIN {X 0,Y 566.145,Z 440.463,A -85,B 0,C 180,E1 -2501.921,E2 -2501.921} C_VEL
LIN {X 0,Y 566.17,Z 440.455,A -85,B 0,C 180,E1 -2504.891,E2 -2504.891} C_VEL
LIN {X 0,Y 566.169,Z 440.462,A -85,B 0,C 180,E1 -2507.819,E2 -2507.819} C_VEL
LIN {X 0,Y 566.144,Z 440.463,A -85,B 0,C 180,E1 -2509.993,E2 -2509.993} C_VEL
LIN {X 0,Y 566.175,Z 440.453,A -85,B 0,C 180,E1 -2512.871,E2 -2512.871} C_VEL
LIN {X 0,Y 566.241,Z 440.446,A -85,B 0,C 180,E1 -2515.017,E2 -2515.017} C_VEL
LIN {X 0,Y 566.271,Z 440.449,A -85,B 0,C 180,E1 -2517.867,E2 -2517.867} C_VEL
LIN {X 0,Y 566.279,Z 440.446,A -85,B 0,C 180,E1 -2520.001,E2 -2520.001} C_VEL
LIN {X 0,Y 566.23,Z 440.447,A -85,B 0,C 180,E1 -2522.847,E2 -2522.847} C_VEL
LIN {X 0,Y 566.228,Z 440.454,A -85,B 0,C 180,E1 -2525.7,E2 -2525.7} C_VEL
LIN {X 0,Y 566.18,Z 440.45,A -85,B 0,C 180,E1 -2528.567,E2 -2528.567} C_VEL
LIN {X 0,Y 566.189,Z 440.452,A -85,B 0,C 180,E1 -2531.456,E2 -2531.456} C_VEL
LIN {X 0,Y 566.199,Z 440.452,A -85,B 0,C 180,E1 -2534.495,E2 -2534.495} C_VEL
LIN {X 0,Y 566.146,Z 440.457,A -85,B 0,C 180,E1 -2537.334,E2 -2537.334} C_VEL
LIN {X 0,Y 566.142,Z 440.46,A -85,B 0,C 180,E1 -2540.341,E2 -2540.341} C_VEL
LIN {X 0,Y 566.156,Z 440.457,A -85,B 0,C 180,E1 -2542.633,E2 -2542.633} C_VEL
LIN {X 0,Y 566.176,Z 440.452,A -85,B 0,C 180,E1 -2545.022,E2 -2545.022} C_VEL
LIN {X 0,Y 566.152,Z 440.455,A -85,B 0,C 180,E1 -2547.343,E2 -2547.343} C_VEL
LIN {X 0,Y 566.155,Z 440.464,A -85,B 0,C 180,E1 -2549.772,E2 -2549.772} C_VEL
LIN {X 0,Y 566.174,Z 440.455,A -85,B 0,C 180,E1 -2552.426,E2 -2552.426} C_VEL
LIN {X 0,Y 566.157,Z 440.455,A -85,B 0,C 180,E1 -2554.987,E2 -2554.987} C_VEL
LIN {X 0,Y 566.18,Z 440.457,A -85,B 0,C 180,E1 -2557.463,E2 -2557.463} C_VEL
LIN {X 0,Y 566.157,Z 440.461,A -85,B 0,C 180,E1 -2560.204,E2 -2560.204} C_VEL
LIN {X 0,Y 566.14,Z 440.458,A -85,B 0,C 180,E1 -2563.061,E2 -2563.061} C_VEL
LIN {X 0,Y 566.152,Z 440.464,A -85,B 0,C 180,E1 -2566.054,E2 -2566.054} C_VEL
LIN {X 0,Y 566.134,Z 440.456,A -85,B 0,C 180,E1 -2568.857,E2 -2568.857} C_VEL
LIN {X 0,Y 566.172,Z 440.46,A -85,B 0,C 180,E1 -2571.636,E2 -2571.636} C_VEL
LIN {X 0,Y 566.134,Z 440.463,A -85,B 0,C 180,E1 -2574.306,E2 -2574.306} C_VEL
LIN {X 0,Y 566.162,Z 440.455,A -85,B 0,C 180,E1 -2576.894,E2 -2576.894} C_VEL
LIN {X 0,Y 566.16,Z 440.46,A -85,B 0,C 180,E1 -2579.406,E2 -2579.406} C_VEL
LIN {X 0,Y 566.137,Z 440.467,A -85,B 0,C 180,E1 -2581.854,E2 -2581.854} C_VEL
LIN {X 0,Y 566.187,Z 440.498,A -85,B 0,C 180,E1 -2584.861,E2 -2584.861} C_VEL
LIN {X 0,Y 566.277,Z 441.038,A -85,B 0,C 180,E1 -2585.041,E2 -2585.041} C_VEL
LIN {X 0,Y 566.914,Z 446.244,A -85,B 0,C 180,E1 -2586.047,E2 -2586.047} C_VEL
LIN {X 0,Y 566.684,Z 462.916,A -85,B 0,C 180,E1 -2589.111,E2 -2589.111} C_VEL
LIN {X 0,Y 566.521,Z 479.472,A -85,B 0,C 180,E1 -2592.119,E2 -2592.119} C_VEL
LIN {X 0,Y 566.319,Z 496.986,A -85,B 0,C 180,E1 -2595.248,E2 -2595.248} C_VEL
LIN {X 0,Y 566.289,Z 501.249,A -85,B 0,C 180,E1 -2595.972,E2 -2595.972} C_VEL
LIN {X 0,Y 566.618,Z 503.437,A -85,B 0,C 180,E1 -2596.045,E2 -2596.045} C_VEL
LIN {X 0,Y 567.16,Z 509.098,A -85,B 0,C 180,E1 -2596.131,E2 -2596.131} C_VEL
